# B&R Automation Studio project 8238 (part 32)

#### _getTourLoadingData.st
```iecst
ACTION _getTourLoadingData:

	prg	:= 0;
	cat := 0;
	cus := 0;
	dst := 0;
	sp1 := 0;
	sp2 := 0;
	sp3 := 0;
	index 	:= 0;
	tourID := 0;

	error := 0;
	found := 0;
	//Set common parameters of the function.
	getParameterName.searchString := requestData;
	getParameterName.searchOffset := 0;
	getParameterName.searchEndProperty := STRING_DOLLAR;

	//Find the index
	getParameterName.searchPropertyName := '"displayId":';
	getParameterName.searchEndProperty := ',';
	getParameterName();
	IF getParameterName.status = ERR_OK THEN
		index := DINT_TO_UDINT(atoi(ADR(getParameterName.outputValue)));
		getParameterName.searchOffset := getParameterName.nextPosition;
	ELSE
		error := 1;
	END_IF;

	//Find the category
	getParameterName.searchPropertyName := '"cat":';
	getParameterName.searchEndProperty := ',';
	getParameterName();
	IF getParameterName.status = ERR_OK THEN
		cat := DINT_TO_UDINT(atoi(ADR(getParameterName.outputValue)));
		getParameterName.searchOffset := getParameterName.nextPosition;
	ELSE
		error := 2;
	END_IF;

	//Find the customer
	getParameterName.searchPropertyName := '"cus":';
	getParameterName.searchEndProperty := ',';
	getParameterName();
	IF getParameterName.status = ERR_OK THEN
		cus := DINT_TO_UDINT(atoi(ADR(getParameterName.outputValue)));
		getParameterName.searchOffset := getParameterName.nextPosition;
	ELSE
		error := 3;
	END_IF;

	//Find the tour
	getParameterName.searchPropertyName := '"tourId":';
	getParameterName.searchEndProperty := ',';
	getParameterName();
	IF getParameterName.status = ERR_OK THEN
		tourID := DINT_TO_UDINT(atoi(ADR(getParameterName.outputValue)));
		getParameterName.searchOffset := getParameterName.nextPosition;
	ELSE
		error := 4;
	END_IF;

	//Find the Program
	getParameterName.searchPropertyName := '"prg":';
	getParameterName.searchEndProperty := ',';
	getParameterName();
	IF getParameterName.status = ERR_OK THEN
		prg := DINT_TO_USINT(atoi(ADR(getParameterName.outputValue)));
		getParameterName.searchOffset := getParameterName.nextPosition;
	ELSE
		error := 5;
	END_IF;

	//Find the sp1
	getParameterName.searchPropertyName := '"sp1":';
	getParameterName.searchEndProperty := ',';
	getParameterName();
	IF getParameterName.status = ERR_OK THEN
		sp1 := DINT_TO_UINT(atoi(ADR(getParameterName.outputValue)));
		getParameterName.searchOffset := getParameterName.nextPosition;
	ELSE
		error := 6;
	END_IF;

	//Find the sp2
	getParameterName.searchPropertyName := '"sp2":';
	getParameterName.searchEndProperty := ',';
	getParameterName();
	IF getParameterName.status = ERR_OK THEN
		sp2 := DINT_TO_UINT(atoi(ADR(getParameterName.outputValue)));
		getParameterName.searchOffset := getParameterName.nextPosition;
	ELSE
		error := 7;
	END_IF;
	//Find the sp3
	getParameterName.searchPropertyName := '"sp3":';
	getParameterName.searchEndProperty := ',';
	getParameterName();
	IF getParameterName.status = ERR_OK THEN
		sp3 := DINT_TO_UINT(atoi(ADR(getParameterName.outputValue)));
		getParameterName.searchOffset := 0;//getParameterName.nextPosition;
	ELSE
		error := 8;
	END_IF;

	//Find the program
	getParameterName.searchPropertyName := '"dst":';
	getParameterName.searchEndProperty := ',';
	getParameterName();
	IF getParameterName.status = ERR_OK THEN
		dst := DINT_TO_USINT(atoi(ADR(getParameterName.outputValue)));
		IF (index <= MAX_DISPLAYS) THEN
			found := found + 1;
			bag ACCESS ADR(LiveData_Recv[index].Bag);
			bag.Cat := cat;
			bag.Prg := prg;
			bag.Cus := cus;
			bag.Dst := dst;
			LiveData_Recv[index].Setpoints.SP1 := sp1 * 10;
			LiveData_Recv[index].Setpoints.SP2:= sp2 * 10;
			LiveData_Recv[index].Setpoints.SP3 := sp3 * 10;
			//bag.Tour := tourID;
		ELSE
			error := 99;
			overRideData.responseHeader.status := '404 Not Found';
			responseData := 'Unknown display';
			httpServer.responseDataLen := LEN(responseData);
		END_IF;
	ELSE
		error := 10;
	END_IF;

	sendResponse := (found > 0);
	errorResponse := (error > 0);

END_ACTION
```

#### _getTourLoadingSubmit.st
```iecst
ACTION _getTourLoadingSubmit:

	prg	:= 0;
	cat := 0;
	cus := 0;
	dst := 0;
	sp1 := 0;
	sp2 := 0;
	sp3 := 0;
	index 	:= 0;
	tourID := 0;

	error := 0;
	found := 0;
	//Set common parameters of the function.
	getParameterName.searchString := requestData;
	getParameterName.searchOffset := 0;
	getParameterName.searchEndProperty := STRING_DOLLAR;

	//Find the index
	getParameterName.searchPropertyName := '"displayId":';
	getParameterName.searchEndProperty := ',';
	getParameterName();
	IF getParameterName.status = ERR_OK THEN
		index := DINT_TO_UDINT(atoi(ADR(getParameterName.outputValue)));
		getParameterName.searchOffset := getParameterName.nextPosition;
	ELSE
		error := 1;
	END_IF;

	//Find the category
	getParameterName.searchPropertyName := '"cat":';
	getParameterName.searchEndProperty := ',';
	getParameterName();
	IF getParameterName.status = ERR_OK THEN
		cat := DINT_TO_UDINT(atoi(ADR(getParameterName.outputValue)));
		getParameterName.searchOffset := getParameterName.nextPosition;
	ELSE
		error := 2;
	END_IF;

	//Find the customer
	getParameterName.searchPropertyName := '"cus":';
	getParameterName.searchEndProperty := ',';
	getParameterName();
	IF getParameterName.status = ERR_OK THEN
		cus := DINT_TO_UDINT(atoi(ADR(getParameterName.outputValue)));
		getParameterName.searchOffset := getParameterName.nextPosition;
	ELSE
		error := 3;
	END_IF;

	//Find the tour
	getParameterName.searchPropertyName := '"tourId":';
	getParameterName.searchEndProperty := ',';
	getParameterName();
	IF getParameterName.status = ERR_OK THEN
		tourID := DINT_TO_UDINT(atoi(ADR(getParameterName.outputValue)));
		getParameterName.searchOffset := getParameterName.nextPosition;
	ELSE
		error := 4;
	END_IF;

	//Find the Program
	getParameterName.searchPropertyName := '"prg":';
	getParameterName.searchEndProperty := ',';
	getParameterName();
	IF getParameterName.status = ERR_OK THEN
		prg := DINT_TO_USINT(atoi(ADR(getParameterName.outputValue)));
		getParameterName.searchOffset := getParameterName.nextPosition;
	ELSE
		error := 5;
	END_IF;

	//Find the sp1
	getParameterName.searchPropertyName := '"sp1":';
	getParameterName.searchEndProperty := ',';
	getParameterName();
	IF getParameterName.status = ERR_OK THEN
		sp1 := DINT_TO_UINT(atoi(ADR(getParameterName.outputValue)));
		getParameterName.searchOffset := getParameterName.nextPosition;
	ELSE
		error := 6;
	END_IF;

	//Find the sp2
	getParameterName.searchPropertyName := '"sp2":';
	getParameterName.searchEndProperty := ',';
	getParameterName();
	IF getParameterName.status = ERR_OK THEN
		sp2 := DINT_TO_UINT(atoi(ADR(getParameterName.outputValue)));
		getParameterName.searchOffset := getParameterName.nextPosition;
	ELSE
		error := 7;
	END_IF;
	//Find the sp3
	getParameterName.searchPropertyName := '"sp3":';
	getParameterName.searchEndProperty := ',';
	getParameterName();
	IF getParameterName.status = ERR_OK THEN
		sp3 := DINT_TO_UINT(atoi(ADR(getParameterName.outputValue)));
		getParameterName.searchOffset := 0;//getParameterName.nextPosition;
	ELSE
		error := 8;
	END_IF;

	//Find the program
	getParameterName.searchPropertyName := '"dst":';
	getParameterName.searchEndProperty := ',';
	getParameterName();
	IF getParameterName.status = ERR_OK THEN
		dst := DINT_TO_USINT(atoi(ADR(getParameterName.outputValue)));
		IF (index <= MAX_DISPLAYS) THEN
			found := found + 1;
			bag ACCESS ADR(LiveData_Recv[index].Bag);
			bag.Cat := cat;
			bag.Prg := prg;
			bag.Cus := cus;
			bag.Dst := dst;
			LiveData_Recv[index].Setpoints.SP1 := sp1 * 10;
			LiveData_Recv[index].Setpoints.SP2:= sp2 * 10;
			LiveData_Recv[index].Setpoints.SP3 := sp3 * 10;
			LiveData_Recv[index].Submit_Loading := 1;

			//bag.Tour := tourID;
		ELSE
			error := 99;
			overRideData.responseHeader.status := '404 Not Found';
			responseData := 'Unknown display';
			httpServer.responseDataLen := LEN(responseData);
		END_IF;
	ELSE
		error := 10;
	END_IF;

	sendResponse := (found > 0);
	errorResponse := (error > 0);

END_ACTION
```

#### Types.typ - Local data types
```iecst
TYPE
	overRide_typ : 	STRUCT  (** OverRide Data to override default setting*)
		responseDataLen : UDINT;
		responseHeader : httpResponseHeader_t;
	END_STRUCT;
END_TYPE
```

#### LocalFunctions.fun
```iecst
FUNCTION_BLOCK httpGetParameter (*FUB to Get parameter values set in URI or BODY...*) (*$GROUP=User,$CAT=User,$GROUPICON=User.png,$CATICON=User.png*)
	VAR_INPUT
		searchPropertyName : STRING[50]; (*StringValue of propery or name to match*)
		searchEndProperty : STRING[50]; (*String Character or value to show end of property value -- DEFAULT & *)
		searchOffset : UINT; (*Offset can be set to skip searching begining of string if not required*)
		searchString : STRING[500];
	END_VAR
	VAR_OUTPUT
		outputValue : STRING[100]; (*String Value found*)
		status : UINT;
		nextPosition : UINT;
	END_VAR
	VAR
		matchString : STRING[50];
		inputData : ARRAY[0..499] OF USINT;
		endIndex : INT;
		startPosition : INT;
		n : INT;
		compare : DINT;
		length : UINT;
		startoffset : UINT;
		search : STRING[50];
	END_VAR
END_FUNCTION_BLOCK
```

#### httpGetParameter.st
```iecst
(* FUB to Get parameter values set in URI or BODY... *)
FUNCTION_BLOCK httpGetParameter
	status := ERR_FUB_BUSY;
// Get the function Name from the URI
//Use the string length of the service name	+
	memset(ADR(outputValue),0,SIZEOF(outputValue));
	matchString := searchPropertyName;
	strcpy(ADR(inputData[0]),ADR(searchString));
	startoffset := searchOffset;
	endIndex := LEN(searchString);
	startPosition := 16#FFF;
	IF endIndex > startoffset THEN
		FOR n := startoffset TO endIndex DO
			memcpy(ADR(search),ADR(inputData[n]),LEN(matchString));
			compare := 	strcmp(ADR(search),ADR(matchString));
			IF (compare = 0) THEN
				startPosition := n + LEN(matchString);
				EXIT;
			END_IF;
		END_FOR;
	ELSE
		status := 100;
	END_IF;

	IF (startPosition <> 16#FFF) THEN
		//Get the End Position
		matchString := searchEndProperty;
		memset(ADR(search),0,SIZEOF(search));
		startoffset := startPosition;
		IF endIndex >= startoffset THEN
			FOR n := startoffset TO endIndex DO
				memcpy(ADR(search),ADR(inputData[n]),LEN(matchString));
				compare := 	strcmp(ADR(search),ADR(matchString));
				length := n - startPosition;
				IF (compare = 0) THEN
					EXIT;
				END_IF;
			END_FOR;
			outputValue := MID(searchString,length,startPosition + 1);
			nextPosition := startPosition + length;
			status := ERR_OK;
		ELSE
			status := 102;
		END_IF;
	ELSE
		outputValue := '';
		nextPosition := 0;
		status := 101;
	END_IF;

END_FUNCTION_BLOCK
```

#### _updateVarByName.st
```iecst
//0, 15// Derived data types Data types declared with the construction TYPE...END_TYPE [1], [2]
//1:// BOOL 8-bit containing a boolean value FALSE=0 OR TRUE=1
//2:// SINT 8-bit signed integer
//3:// INT 16-bit signed integer
//4:// DINT 32-bit signed integer
//5:// USINT 8-bit unsigned integer
//6:// UINT 16-bit unsigned integer
//7:// UDINT 32-bit unsigned integer
//8:// REAL 32-bit floating point number
//9:// STRING Variable-length single-byte character string
//10:// ULINT 	64-bit unsigned integer
//11:// DATE_AND_TIME 32-bit date in seconds since 01/01/1970 00:00:00
//12:// TIME 32-bit time in ms
//13:// DATE 32-bit date (only)
//14:// LREAL 64-bit floating point number
//16:// TIME_OF_DAY 32-bit time OF day (only)
//17:// BYTE 	Bit string OF length 8
//18:// WORD Bit string OF length 16
//19:// DWORD Bit string OF length 32
//20:// LWORD Bit string OF length 64
//21:// WSTRING Variable-length double-byte character string
//23:// LINT 	64-bit signed integer

ACTION _updateVarByName:

//{"varName":"xxx","value":10}
//{"varName":"xxx","value":"stringValue"}
scanCount := 0;
WHILE (scanCount <= 19) AND NOT sendResponse AND NOT errorResponse DO
	scanCount := scanCount + 1; //Supercharge peformance by doing 20 scans per cycle

	CASE setValue OF

		0:// init search vars
			searchOffset := 0;
			//Create a FIFO to write our values into so we can commit them on success!!
			arrayEnd := FIND(requestData,'}]');// Be sure to check for end ] or we could get errors updating arrays.
			error := 0;
			setValue := 1;
			pos1 := 0;
			pos2 := 0;

		1:// create fifo to write data into.
			createFifo.enable := 1;
			createFifo.mode := fifoMODE_WRITE_UNTIL_FULL;
			createFifo.size := LEN(requestData);
			createFifo.pFifo := ADR('update-by-name-list');
			createFifo();
			IF (createFifo.status = ERR_OK) THEN
				setValue := 4;
			ELSIF (createFifo.status = fifoERR_FIFO_ALREADY_EXISTS) THEN
				setValue := 2;
			ELSIF (createFifo.status <> ERR_FUB_BUSY) THEN
				setValue := 100;
				status := 94;
			END_IF;

		2:// get ident if fifo already exists
			fi_status := fifoGetIdent(createFifo.pFifo,ADR(createFifo.ident));
			IF fi_status = ERR_OK THEN
				setValue := 3;
			ELSE
				setValue := 100;
				status := 94;
			END_IF;

		3:// Clear the FIFO if it already exists
			clearFifo.enable := 1;
			clearFifo.ident := createFifo.ident;
			clearFifo();
			IF clearFifo.status = ERR_OK THEN
				setValue := 4;
			ELSIF (clearFifo.status <> ERR_FUB_BUSY) THEN
				setValue := 100;
				status := 94;
			END_IF;

		4:// Validate the json, make sure if we have a [
			IF (arrayEnd > 0) THEN
				IF FIND(requestData,'[{') > 0 THEN
					setValue := 5; //Array start and end found
				ELSE
					setValue := 100;
					status := 95;
				END_IF;
			ELSE
				IF FIND(requestData,'[{') = 0 THEN
					setValue := 5; //Array start and end not found
				ELSE
					setValue := 100;
					status := 95;
				END_IF;
			END_IF;

		5://find the order of the parameters in the request sting.
			found 	:= 0;
			getParameterName.searchString := requestData;
			IF (pos1 = 0) THEN
				pos1 := FIND(requestData,SEARCH_STRING_VAR_NAME);
				pos2 := FIND(requestData,SEARCH_STRING_VAR_VALUE);
			END_IF;
			IF (pos1 = 0) OR (pos2 = 0) THEN
				setValue := 100;
				status := 93;
			ELSIF (pos1 > pos2) THEN
				setValue := 6;
			ELSE
				setValue := 8;
			END_IF;

		6:// find the value first
			value 	:= '';
			isString := 0;
			getParameterName.searchPropertyName := SEARCH_STRING_VAR_VALUE;
			getParameterName.searchEndProperty := ',';
			getParameterName.searchOffset := searchOffset;
			getParameterName();
			IF getParameterName.status = ERR_OK THEN
				searchOffset := getParameterName.nextPosition;
				//If we have been passed a string remove the ""
				IF LEFT(getParameterName.outputValue,1) = '"' THEN
					isString := 1;
					value := MID(getParameterName.outputValue,(LEN(getParameterName.outputValue) - 2),2);
				ELSE
					value := getParameterName.outputValue;
				END_IF;
				setValue := 7;
			ELSE
				setValue := 100;
				status := 2;
			END_IF;

		7:// find the name 2nd
			varName := '';
			found 	:= 0;
			//Set common parameters of the function.

			getParameterName.searchOffset := searchOffset;
			//Find the id
			getParameterName.searchPropertyName := SEARCH_STRING_VAR_NAME;
			getParameterName.searchEndProperty := '"';
			getParameterName();
			IF getParameterName.status = ERR_OK THEN
				varName := getParameterName.outputValue;
				searchOffset := getParameterName.nextPosition;
				setValue := 10;
			ELSE
				setValue := 100;
				status := 1;
			END_IF;

		8:// find the first param

			varName := '';
			getParameterName.searchOffset := searchOffset;
			//Find the id
			getParameterName.searchPropertyName := SEARCH_STRING_VAR_NAME;
			getParameterName.searchEndProperty := '"';
			getParameterName();
			IF getParameterName.status = ERR_OK THEN
				varName := getParameterName.outputValue;
				searchOffset := getParameterName.nextPosition;
				setValue := 9;
			ELSE
				setValue := 100;
				status := 1;
			END_IF;

		9:// find the 2nd param
			value 	:= '';
			isString := 0;
			getParameterName.searchPropertyName := SEARCH_STRING_VAR_VALUE;
			getParameterName.searchEndProperty := '}';
			getParameterName.searchOffset := searchOffset;
			getParameterName();
			IF getParameterName.status = ERR_OK THEN
				searchOffset := getParameterName.nextPosition;
				//If we have been passed a string remove the ""
				IF LEFT(getParameterName.outputValue,1) = '"' THEN
					isString := 1;
					value := MID(getParameterName.outputValue,(LEN(getParameterName.outputValue) - 2),2);
				ELSE
					value := getParameterName.outputValue;
				END_IF;
				setValue := 10;
			ELSE
				setValue := 100;
				status := 2;
			END_IF;

		10: //get the ident

			//status := PV_ident(ADR(varName),1,0,ADR(ident));
			status := PV_xgetadr(ADR(varName),ADR(pv_adr),ADR(pv_len));
			IF (status = ERR_OK) THEN
				setValue := 11;
			ELSIF (status <> ERR_FUB_BUSY) THEN
				IF (status = 14710) THEN
					overRideData.responseHeader.status := '404 Not Found';
					responseData := 'PV Not found';
					httpServer.responseDataLen := LEN(responseData);
				END_IF;
				setValue := 100;//
			END_IF;

		11: // Get the data type so we can scale correctly
			status := PV_ninfo(ADR(varName),ADR(pv_type),ADR(pv_length),ADR(pv_dimension));
			IF (status = ERR_OK) THEN
				setValue := 12;
			ELSIF (status <> ERR_FUB_BUSY) THEN
				setValue := 100;//
			END_IF;

		12: // Found update the value
			//Type 0 or 15 is part of a type not a var name.
			//We must also check the dimension is 1 or we are trying to update the root of an array.
			//TEMP INCASE OF MALFORM JSON
			//			IF (isString AND (pv_type <> 9)) THEN
			//				isString := 0;
			//			END_IF;

			stringCheck := (NOT isString AND (pv_type <> 9)) OR (isString AND (pv_type = 9)); // We have to modify this if we want to support strings other than STRING
			IF (pv_dimension = 1) AND stringCheck THEN
				num_Val := atoi(ADR(value));
				CASE pv_type OF
					0,15:// Derived data types Data types declared with the construction TYPE...END_TYPE [1], [2]
						status := 99;
						setValue := 100;
					1:// BOOL
						IF (num_Val >= 0) AND (num_Val <= 1) THEN
							pData := ADR(num_Val);
							//memcpy(pv_adr,ADR(num_Val),pv_length);
							found := 1;
						ELSE
							status := 96;
							setValue := 100;
						END_IF;
					2:// SINT
						IF (num_Val >= -128) AND (num_Val <= 16#7F) THEN
							pData := ADR(num_Val);
							//memcpy(pv_adr,ADR(num_Val),pv_length);
							found := 1;
						ELSE
							status := 96;
							setValue := 100;
						END_IF;
					3:// INT
						IF (num_Val >= -32768) AND (num_Val <= 16#7FFF) THEN
							pData := ADR(num_Val);
							//memcpy(pv_adr,ADR(num_Val),pv_length);
							found := 1;
						ELSE
							status := 96;
							setValue := 100;
						END_IF;
					4:// DINT
						IF (num_Val >= -2147483648) AND (num_Val <= 16#7FFFFFFF) THEN
							pData := ADR(num_Val);
							//memcpy(pv_adr,ADR(num_Val),pv_length);
							found := 1;
						ELSE
							status := 96;
							setValue := 100;
						END_IF;

					5: //USINT
						IF (num_Val >= 0) AND (num_Val <= 16#FF) THEN
							pData := ADR(num_Val);
							//memcpy(pv_adr,ADR(num_Val),pv_length);
							found := 1;
						ELSE
							status := 96;
							setValue := 100;
						END_IF;
					6:// UINT
						IF (num_Val >= 0) AND (num_Val <= 16#FFFF) THEN
							pData := ADR(num_Val);
							//memcpy(pv_adr,ADR(num_Val),pv_length);
							found := 1;
						ELSE
							status := 96;
							setValue := 100;
						END_IF;
					7: //UDINT
						IF (num_Val >= 0) AND (DINT_TO_UDINT(num_Val) <= 16#FFFF_FFFF) THEN  //
							pData := ADR(num_Val);
							//memcpy(pv_adr,ADR(num_Val),pv_length);
							found := 1;
						ELSE
							status := 96;
							setValue := 100;
						END_IF;

					8:// REAL 32-bit floating point number
						float_val := atof(ADR(value));
						IF (float_val >= -3.4E38) AND (float_val <= 3.4E38) THEN
							pData := ADR(float_val);
							//memcpy(pv_adr,ADR(float_val),pv_length);
							found := 1;
						ELSE
							status := 96;
							setValue := 100;
						END_IF;
						found := 1;

					9:// STRING Variable-length single-byte character string
						IF (LEN(value) <= pv_length) THEN
							memset(ADR(string_Val),0,pv_length);
							memcpy(ADR(string_Val),ADR(value),LEN(value));
							pData := ADR(string_Val);
							found := 1;
						ELSE
							status := 96;
							setValue := 100;
						END_IF;
					10..14,16..23:
						status := 98;
						setValue := 100;

				END_CASE;
			ELSIF NOT stringCheck THEN
				status := 97;
				setValue := 100;
			ELSE;
				status := 99;
				setValue := 100;
			END_IF;
			IF (found > 0) THEN
				setValue := 13;
			END_IF;

		13: // Add header data to the fifo
			data[0] := pv_adr;
			data[1] := pv_len;
			writeFifo.enable := 1;
			writeFifo.ident := createFifo.ident;
			writeFifo.pData := ADR(data[0]);
			writeFifo.size := 8;//
			writeFifo();
			IF (writeFifo.status = ERR_OK) THEN
				setValue := 14;
			ELSIF writeFifo.status <> ERR_FUB_BUSY THEN
				setValue := 100;
				status := 94;
			END_IF;

		14:// Add the actual data the fifo
			writeFifo.enable := 1;
			writeFifo.ident := createFifo.ident;
			writeFifo.pData := pData;
			writeFifo.size := pv_len;//
			writeFifo();
			IF (writeFifo.status = ERR_OK) THEN
				setValue := 20;
			ELSIF writeFifo.status <> ERR_FUB_BUSY THEN
				setValue := 100;
				status := 94;
			END_IF;

		20:// Check if we need to search again or complete the
			IF(arrayEnd <= 1) OR ((arrayEnd - searchOffset) < 5) THEN
				setValue := 30;
			ELSE //Search again
				setValue := 5;
			END_IF;

		30:// Process the results Read out the data header
			readFifo.enable := 1;
			readFifo.ident := createFifo.ident;
			readFifo.pData := ADR(data[0]);
			readFifo.size := 8;
			readFifo();
			IF (readFifo.status = ERR_OK) THEN
				pv_adr := data[0];
				pv_len := data[1];
				setValue := 31;
			ELSIF (readFifo.status = fifoERR_BUFFER_EMPTY) THEN
				setValue := 40;
			ELSIF readFifo.status <> ERR_FUB_BUSY THEN
				setValue := 100;
				status := 94;
			END_IF;

		31:// Process the results Read out the data
			readFifo.enable := 1;
			readFifo.ident := createFifo.ident;
			readFifo.pData := pv_adr;
			readFifo.size := pv_len;
			readFifo();
			IF (readFifo.status = ERR_OK) THEN
				setValue := 30; // Go back to iterate through the fifo
				//			ELSIF (readFifo.status = fifoERR_BUFFER_EMPTY) THEN
				//				setValue := 40;
			ELSIF readFifo.status <> ERR_FUB_BUSY THEN
				setValue := 100;
				status := 94;
			END_IF;

		40:// Delete the FIFO
			deleteFifo.enable := 1;
			deleteFifo.ident := createFifo.ident;
			deleteFifo();
			IF deleteFifo.status = ERR_OK THEN
				setValue := 90;
			ELSIF (deleteFifo.status <> ERR_FUB_BUSY) THEN
				setValue := 100;
				status := 94;
			END_IF;

		90:// Send the response

		100:// Error Step
			error := status;

			CASE status OF
				94:
					overRideData.responseHeader.status := '400 Bad Request';
					responseData := 'PLC FIFO Failure';
					httpServer.responseDataLen := LEN(responseData);

				95:
					overRideData.responseHeader.status := '400 Bad Request';
					responseData := 'Malformed JSON array';
					httpServer.responseDataLen := LEN(responseData);

				96:
					overRideData.responseHeader.status := '403 Forbidden';
					responseData := 'Value out of range';
					httpServer.responseDataLen := LEN(responseData);

				97:
					overRideData.responseHeader.status := '405 Method Not Allowed';
					responseData := 'You have sent a string to a numeric data type';
					httpServer.responseDataLen := LEN(responseData);

				98:
					overRideData.responseHeader.status := '405 Method Not Allowed';
					responseData := 'This data type is currently not supported';
					httpServer.responseDataLen := LEN(responseData);
				99:
					overRideData.responseHeader.status := '403 Forbidden';
					responseData := 'You have requested to update a structure part, or Array item without specifing the full path';
					httpServer.responseDataLen := LEN(responseData);
			END_CASE;

	END_CASE;

	sendResponse := (setValue = 90);
	errorResponse := (error > 0);
	//Configuration.Data.Belt[0].Alarm.General
	IF EDGEPOS(sendResponse) OR EDGEPOS(errorResponse) THEN
		setValue := 0;
	END_IF;
END_WHILE;

END_ACTION
```

#### _nedlinSetCustomer.st
```iecst
ACTION _nedlinSetCustomer:
	//{"stationId":1,"cus":25}
	IF (found = 0) AND (error = 0) THEN
		index := 0;
		cus := 0;

		error := 0;
		found := 0;
		//Set common parameters of the function.
		getParameterName.searchString := requestData;
		getParameterName.searchOffset := 0;
		getParameterName.searchEndProperty := STRING_DOLLAR;

		//Find the Index
		getParameterName.searchPropertyName := '"stationId":';
		getParameterName.searchEndProperty := ',';
		getParameterName();
		IF getParameterName.status = ERR_OK THEN
			index := DINT_TO_UDINT(atoi(ADR(getParameterName.outputValue)));
		ELSE
			error := 2;
		END_IF;

		//Find the customer
		getParameterName.searchPropertyName := '"cus":';
		getParameterName.searchEndProperty := ',';
		getParameterName();
		IF getParameterName.status = ERR_OK THEN
			cus := DINT_TO_USINT(atoi(ADR(getParameterName.outputValue)));
			IF (index >= 0) AND (index <= 1) THEN
				CSP[index].Customer := cus;
				found := found + 1;
			ELSE
				error := 99;
				overRideData.responseHeader.status := '404 Not Found';
				responseData := 'Index out of range';
				httpServer.responseDataLen := LEN(responseData);
			END_IF;
		ELSE
			error := 3;
		END_IF;
	END_IF;

	sendResponse := (found > 0);
	errorResponse := (error > 0);

END_ACTION
```

#### _resetCount.st
```iecst
ACTION _resetCount:
	//{"id":1}
	IF (found = 0) AND (error = 0) THEN
		index := 0;
		cus := 0;

		error := 0;
		found := 0;
		//Set common parameters of the function.
		getParameterName.searchString := requestData;
		getParameterName.searchOffset := 0;
		getParameterName.searchEndProperty := STRING_DOLLAR;

		//Find the Index
		getParameterName.searchPropertyName := '"id":';
		getParameterName.searchEndProperty := '}';
		getParameterName();
		IF getParameterName.status = ERR_OK THEN
			index := DINT_TO_UDINT(atoi(ADR(getParameterName.outputValue)));
			IF (index >= 0) AND (index <= MAX_STATIONS) THEN
				SortingBins.counting_frames[index].count := 0;
				found := found + 1;
			ELSE
				error := 99;
				overRideData.responseHeader.status := '404 Not Found';
				responseData := 'Index out of range';
				httpServer.responseDataLen := LEN(responseData);
			END_IF;

		ELSE
			error := 2;
		END_IF;
	END_IF;

	sendResponse := (found > 0);
	errorResponse := (error > 0);

END_ACTION
```

### HttpInstances.txt
```
List Of HTTP_Comm indexes

01: zzReportsHttp
02: SLX_Inteface
03: Configuration
04: OPCuA_Connect
05: Bag Maintenance
06:
07:
08:
09:
10:
11:
12:
13:
14:
15:
16:
17:
18:
19:
20:
```

### Program Logical/http_Lib/zzHttpDriver (IEC, version 3.00.8)

#### Types.typ - Local data types
```iecst
TYPE
	httpState_enum :
		(
		HTTP_CLIENT_WAIT_FOR_COMMAND := 0,
		HTTP_CLIENT_PROCESS_REQUEST := 1,
		HTTP_CLIENT_PROCESS_ENABLE := 2,
		HTTP_CLIENT_PROCESS_SEND := 3,
		HTTP_CLIENT_PROCESS_WAIT_RESP := 4,
		HTTP_CLIENT_PROCESS_RESPONSE := 5,
		HTTP_CLIENT_COMPLETE := 6,
		HTTP_CLIENT_ABORT := 99
		);
END_TYPE
```

#### Variables.var - Local variables
```iecst
VAR
	n : UINT;
	r : UINT;
	httpComm : REFERENCE TO http_comm_typ;
	ringBuffer : ARRAY[0..HTTP_MAX_COMM] OF UINT;
	sizeRingArray : UDINT;
	sizeRingData : UDINT;
	moveSize : UDINT;
	pUrl : UDINT;
	URL : STRING[500];
	pHost : UDINT;
	pResponseHeader : UDINT;
	pTempMem : UDINT;
	sizeTempMem : UDINT;
	pStatistics : UDINT;
	responseHeader : httpResponseHeader_t;
	http_Client : httpClient;
	Statistics : {REDUND_UNREPLICABLE} httpStatistics_t;
	emptyResponseHeader : httpResponseHeader_t;
	DebugErrCount : UDINT;
	pRequestHeader : UDINT;
	requestHeader : httpRequestHeader_t;
	remainingStringLen : DINT;
END_VAR
VAR CONSTANT
	BLANK_CHARACTER : STRING[80] := '';
END_VAR
VAR
	httpState : httpState_enum;
	retryCount : USINT;
	status : HTTP_Status_enum;
	lastError : STRING[60];
	replyCode : UINT;
	count : UDINT;
	testEnable : BOOL;
	testAbort : BOOL;
END_VAR
```

#### Main.st - Init, cyclic, exit code
```iecst
//V2.00.1- First Release of Version Control - Remove all unused code- Removed temp memory for recieve data as this helps when we get a "Invalid Character error"
//V2.00.2 -- ADD: New error handling if we do not recieve data when expected.
//V2.00.3 -- ADD: Add http reply code to the http data type so we don;t have to decode the string in the user tasks
//V3.00.1 -- CHANGE: TR 23/08/2019 - Convert the driver to a state machine
//V3.00.2 -- FIX: When writing to reports the status is being set as disabled causing repeated writes -- Comment out in HTTP_CLIENT_PROCESS_REQUEST and it works.. It makes no sense!!
//V3.00.3 -- FIX: Found solution to 3.02. The original state was being set to DISABLE so the proces step was exiting incorrectly.
//V3.00.4 -- FIX: Issue with certain errors getting stuck on the abort step.
//V3.00.5 -- FIX: 35560 error non more idents availble!!
//V3.00.6 -- FIX: URL Wasn;t not being cleared correctly
//V3.00.7 -- FIX: TCP ERROR could lock up the driver.
//V3.00.8 -- FIX: The way we were passing the http port mean that it was always being set to 0 reegardless of the default setting, when not using overwrite
PROGRAM _INIT
	//Use Static code now but change to config file later..
	HTTP_Config.Host := '10.8.4.220';
	HTTP_Config.Port := 0;
	httpComm ACCESS ADR(HTTP_Comm[0]);

	pUrl 							:= ADR(URL);
	pRequestHeader 					:= ADR(requestHeader);
	pResponseHeader 				:= ADR(responseHeader);
	pStatistics 					:= ADR(Statistics);
	pHost 							:= ADR(requestHeader.host);

	http_Client.pUri 				:= pUrl;
	http_Client.option 				:= httpOPTION_HTTP_11;
	http_Client.pHost 				:= pHost;
	http_Client.pRequestHeader 		:= pRequestHeader;
	http_Client.pResponseHeader 	:= pResponseHeader;
	http_Client.pStatistics 		:= pStatistics;

	//Configure RequestHeader
	requestHeader.protocol := DEFAULT_REQUEST_HEADER.protocol; //'HTTP/1.1';
	requestHeader.contentType := DEFAULT_REQUEST_HEADER.contentType;//'text/plain';
	requestHeader.connection := DEFAULT_REQUEST_HEADER.connection;//'close';
	requestHeader.keepAlive := DEFAULT_REQUEST_HEADER.keepAlive;//'max=100,timeout=5';

	sizeTempMem := 500000; //Allocate 500k of free memory
	TMP_alloc(sizeTempMem,ADR(pTempMem));

	ringBuffer[0] := 0;
	//Check for any requests that were being processed on shut down..
	FOR n := 1 TO HTTP_MAX_COMM DO
		IF HTTP_Comm[n].Status = HTTP_COMM_STATUS_IN_PROCESS THEN
			ringBuffer[0] := n;
		ELSIF HTTP_Comm[n].Status = HTTP_COMM_STATUS_IN_BUFFER THEN
			ringBuffer[n] := n;
		END_IF;
	END_FOR;
	_orderRing;
END_PROGRAM

PROGRAM _CYCLIC

	//Listen to requests and add to ring buffer.
	_ringBuffer;
	http_Client.send	:= EDGEPOS(httpState = HTTP_CLIENT_PROCESS_SEND );
	http_Client.abort	:= EDGEPOS(httpState = HTTP_CLIENT_ABORT);

	CASE httpState OF

		HTTP_CLIENT_WAIT_FOR_COMMAND: // Order the ring buffer and wait for a new command to be processed.
			http_Client.enable := 0;
			retryCount := 0;
			httpComm ACCESS ADR(HTTP_Comm[0]);
			//Wait for next command from ring buffer
			IF(ringBuffer[0] = 0) AND (ringBuffer[1] > 0) THEN
				ringBuffer[0] := ringBuffer[1];
				httpComm ACCESS ADR(HTTP_Comm[ringBuffer[0]]);
				httpComm.Status := HTTP_COMM_STATUS_IN_PROCESS;
				ringBuffer[1] := 0;
			ELSIF (ringBuffer[0] > 0) THEN
				httpState := HTTP_CLIENT_PROCESS_REQUEST;
			END_IF;

		HTTP_CLIENT_PROCESS_REQUEST:
			http_Client.enable := 0;

			replyCode := 0;
			status := HTTP_COMM_STATUS_IN_PROCESS;
			lastError := '';

			httpComm ACCESS ADR(HTTP_Comm[ringBuffer[0]]);

			//brsmemcpy(ADR(URL),ADR(BLANK_CHARACTER),SIZEOF(URL));
			brsmemset(ADR(URL),0,SIZEOF(URL));
			//URL := '';
			brsmemcpy(ADR(URL),httpComm.Command.Cmd_URL.Adr,httpComm.Command.Cmd_URL.Size);
			responseHeader := emptyResponseHeader;

			//Check for any overwrite of the host or header
			IF httpComm.Overwrite.RequestHeader THEN
				requestHeader.protocol 		:= httpComm.Overwrite.RequestHeader_Data.protocol;
				requestHeader.contentType 	:= httpComm.Overwrite.RequestHeader_Data.contentType;
				requestHeader.connection 	:= httpComm.Overwrite.RequestHeader_Data.connection;
				requestHeader.keepAlive 	:= httpComm.Overwrite.RequestHeader_Data.keepAlive;
			ELSE
				requestHeader.protocol 		:= DEFAULT_REQUEST_HEADER.protocol; //'HTTP/1.1';
				requestHeader.contentType 	:= DEFAULT_REQUEST_HEADER.contentType;//'text/plain';
				requestHeader.connection 	:= DEFAULT_REQUEST_HEADER.connection;//'close';
				requestHeader.keepAlive 	:= DEFAULT_REQUEST_HEADER.keepAlive;//'max=100,timeout=5';
			END_IF;
			IF httpComm.Overwrite.Host THEN
				requestHeader.host 		:= httpComm.Overwrite.Host_Config.Host;
				http_Client.hostPort  	:= httpComm.Overwrite.Host_Config.Port;
			ELSE
				requestHeader.host 		:= HTTP_Config.Host;
				http_Client.hostPort 	:= HTTP_Config.Port;
			END_IF;

			requestHeader.contentLength 	:= httpComm.Command.Body_Data.Size;
			http_Client.method 				:= httpComm.Command.Method;
			http_Client.pRequestData 		:= httpComm.Command.Body_Data.Adr;
			http_Client.requestDataLen 		:= httpComm.Command.Body_Data.Size;

			IF (httpComm.Command.ResponseData.Adr > 0) AND (httpComm.Command.ResponseData.Size > 0) THEN
				http_Client.pResponseData 	:= httpComm.Command.ResponseData.Adr;
				http_Client.responseDataSize := httpComm.Command.ResponseData.Size;
			ELSE
				http_Client.pResponseData := pTempMem;
				http_Client.responseDataSize := sizeTempMem;
			END_IF;
			IF (http_Client.status = ERR_FUB_ENABLE_FALSE) AND (http_Client.phase = httpPHASE_NOT_CONNECTED) THEN
				httpState := HTTP_CLIENT_PROCESS_ENABLE;
			END_IF;

		HTTP_CLIENT_PROCESS_ENABLE:
			http_Client.enable := 1;
			IF (http_Client.status = ERR_OK) THEN
				CASE http_Client.phase OF
					httpPHASE_NOT_CONNECTED,httpPHASE_WAITING:
						httpState := HTTP_CLIENT_PROCESS_SEND;

					httpPHASE_SENDING,httpPHASE_RECEIVING:
						httpState := HTTP_CLIENT_PROCESS_WAIT_RESP;

					httpPHASE_RECEIVED:
						httpState := HTTP_CLIENT_PROCESS_SEND; // Received is the left over from the last successful send.
				END_CASE;
			END_IF;

		HTTP_CLIENT_PROCESS_SEND:
			http_Client.enable := 1;
			IF (http_Client.phase = httpPHASE_SENDING) THEN
				httpState := HTTP_CLIENT_PROCESS_WAIT_RESP;
			ELSIF (http_Client.status <> ERR_OK) AND (http_Client.status <> ERR_FUB_BUSY) THEN
				httpState := HTTP_CLIENT_ABORT;
			ELSIF (http_Client.phase = httpPHASE_RECEIVED) AND (http_Client.httpStatus > 0) THEN
				httpState := HTTP_CLIENT_PROCESS_RESPONSE;
			END_IF;

		HTTP_CLIENT_PROCESS_WAIT_RESP:
			http_Client.enable := 1;
			IF (http_Client.phase = httpPHASE_RECEIVED) THEN
				httpState := HTTP_CLIENT_PROCESS_RESPONSE;
			ELSIF (http_Client.status <> ERR_OK) AND (http_Client.status <> ERR_FUB_BUSY) THEN
				httpState := HTTP_CLIENT_ABORT;
			END_IF;

		HTTP_CLIENT_PROCESS_RESPONSE:
			http_Client.enable := 1;
			IF (http_Client.status = ERR_OK) THEN
				replyCode := http_Client.httpStatus;
				CASE http_Client.httpStatus OF
					200..207:
						IF (responseHeader.contentLength > 0) THEN
							IF (responseHeader.contentLength <= httpComm.Command.ResponseData.Size) THEN
								status := HTTP_COMM_STATUS_COMPLETE;
							ELSE
								status := HTTP_COMM_STATUS_ERROR;
								lastError := 'Response data area to small';
							END_IF;
						ELSIF ((httpComm.Command.Method = httpMETHOD_POST) OR (httpComm.Command.Method = httpMETHOD_PUT)) THEN
							status := HTTP_COMM_STATUS_COMPLETE;
						END_IF;
					300..307:
						//Implementation not done
						status := HTTP_COMM_STATUS_ERROR;
						lastError := responseHeader.status;
					400..426: //Errors
						status := HTTP_COMM_STATUS_ERROR;
						lastError := responseHeader.status;
					500..510://Server Errors
						status	:= HTTP_COMM_STATUS_ERROR;
						lastError 	:= responseHeader.status;
					ELSE
						httpState 	:= HTTP_CLIENT_ABORT;
				END_CASE;
			ELSIF (http_Client.status = httpERR_BUFFER_SIZE) THEN	// Response buffer is too small -- Abort and try again with temp memory area

			ELSIF (http_Client.status <> ERR_FUB_BUSY) THEN	//http client failure.
				itoa(http_Client.status,ADR(lastError));
				httpState := HTTP_CLIENT_ABORT;
			END_IF;

			IF (status <> HTTP_COMM_STATUS_IN_PROCESS) THEN
				httpState := HTTP_CLIENT_COMPLETE;
			END_IF;

		HTTP_CLIENT_COMPLETE:
			count := count + 1;
			http_Client.enable := 0;
			httpComm.Status := status;
			httpComm.LastError := lastError;
			httpComm.ReplyCode := replyCode;
			ringBuffer[0] := 0;
			httpState := HTTP_CLIENT_WAIT_FOR_COMMAND;

		HTTP_CLIENT_ABORT:
			http_Client.enable := 1;

			IF ((http_Client.status = ERR_OK) AND NOT http_Client.abort) THEN
				IF (http_Client.phase = httpPHASE_WAITING) OR (http_Client.phase = httpPHASE_NOT_CONNECTED)  THEN
					IF (retryCount > 0) THEN
						httpState := HTTP_CLIENT_COMPLETE;
						status := HTTP_COMM_STATUS_ERROR;
					ELSE
						retryCount := 1;
						httpState := HTTP_CLIENT_PROCESS_REQUEST;
					END_IF;
				ELSIF (http_Client.phase = httpPHASE_RECEIVED) THEN //???
					IF (retryCount > 0) THEN
						httpState := HTTP_CLIENT_COMPLETE;
						status := HTTP_COMM_STATUS_ERROR;
					ELSE
						retryCount := 1;
						httpState := HTTP_CLIENT_PROCESS_REQUEST;
					END_IF;
				END_IF;
			END_IF;
	END_CASE;

	http_Client();

END_PROGRAM
PROGRAM _EXIT
	WHILE (http_Client.status <> ERR_OK) DO
		http_Client.enable := 1;
		http_Client.abort := 1;
		http_Client();
	END_WHILE;

END_PROGRAM
```

#### _ringBuffer.st
```iecst
ACTION _ringBuffer:

	//Listen to new comm events..
	FOR n := 0 TO HTTP_MAX_COMM DO
		//httpComm ACCESS ADR(HTTP_Comm[n]);
		//There is an active comm that is not in the buffer...
		IF (HTTP_Comm[n].Status = HTTP_COMM_STATUS_ACTIVE_WAIT_BUF) THEN
			_addToRing;	//Add to the next avaible space in the ring buffer.
		END_IF;
	END_FOR;

	//Update the ring to ensure we clear any comms that are in error or complete.
	//If a comm is in error, it should be upto the requesting task to clear the error and retry to comm..
	_orderRing;

END_ACTION
```

#### _addToRing.st
```iecst
ACTION _addToRing:
	FOR r := 1 TO HTTP_MAX_COMM DO
		IF (ringBuffer[r] = 0) THEN
			ringBuffer[r] := n;
			HTTP_Comm[n].Status := HTTP_COMM_STATUS_IN_BUFFER;
			EXIT;
		END_IF;
	END_FOR;
END_ACTION
```

#### _orderRing.st
```iecst
ACTION _orderRing:
	//Only loop from position 1 as 0 will be active..
	FOR n := 1 TO HTTP_MAX_COMM DO
		r := ringBuffer[n];
		//If the comm is in not in the queue, or in process then remove it from the queue.
		IF (HTTP_Comm[r].Status <> HTTP_COMM_STATUS_IN_BUFFER)  THEN
			ringBuffer[n] := 0;
		END_IF;
	END_FOR;
	//Shuffle List
	FOR n:= 1 TO (HTTP_MAX_COMM - 1)DO
		IF ringBuffer[n] = 0 THEN
			sizeRingArray := SIZEOF(ringBuffer);
			sizeRingData := SIZEOF(ringBuffer[0]);
			moveSize := (sizeRingArray - ((n+1)*sizeRingData));
			memcpy(ADR(ringBuffer[n]),ADR(ringBuffer[n + 1]),moveSize);
			ringBuffer[HTTP_MAX_COMM] := 0;
		END_IF;
	END_FOR
END_ACTION
```

### Program Logical/LOADCELLS (IEC, version 1.00.1) - LOADCELLS

#### LOADCELLS.st
```iecst
(********************************************************************
 * Program: LOADCELLS
 * File: LOADCELLS.st
 ********************************************************************)
PROGRAM _CYCLIC
(********************************************************************
* ALL SERVOS WITHIN A GROUP MUST HAVE ASCENDING RAIL ID'S
 ********************************************************************)
//	weight1 := DINT_TO_UINT(ABS(WeightRaw[1301].Wgt_Channel_1)/100);
//	weight2 := DINT_TO_UINT(ABS(WeightRaw[1302].Wgt_Channel_1)/100);
//	weight3 := DINT_TO_UINT(ABS(WeightRaw[1303].Wgt_Channel_1)/100);
//	weight4 := DINT_TO_UINT(ABS(WeightRaw[1304].Wgt_Channel_1)/100);
//	weight5 := DINT_TO_UINT(ABS(WeightRaw[1305].Wgt_Channel_1)/100);
//	weight6 := DINT_TO_UINT(ABS(WeightRaw[1306].Wgt_Channel_1)/100);
//	weight7 := DINT_TO_UINT(ABS(WeightRaw[1307].Wgt_Channel_1)/100);
//	weight8 := DINT_TO_UINT(ABS(WeightRaw[1308].Wgt_Channel_1)/100);
//	weight9 := DINT_TO_UINT(ABS(WeightRaw[1309].Wgt_Channel_1)/100);
//	weight10 := DINT_TO_UINT(ABS(WeightRaw[1310].Wgt_Channel_1)/100);
//	weight11 := DINT_TO_UINT(ABS(WeightRaw[1311].Wgt_Channel_1)/100);
//	weight12 := DINT_TO_UINT(ABS(WeightRaw[1312].Wgt_Channel_1)/100);
//	weight13 := DINT_TO_UINT(ABS(WeightRaw[1313].Wgt_Channel_1)/100);
//	weight14 := DINT_TO_UINT(ABS(WeightRaw[1314].Wgt_Channel_1)/100);
//	weight15 := DINT_TO_UINT(ABS(WeightRaw[1315].Wgt_Channel_1)/100);
//	weight16 := DINT_TO_UINT(ABS(WeightRaw[1316].Wgt_Channel_1)/100);
//	weight17 := DINT_TO_UINT(ABS(WeightRaw[1317].Wgt_Channel_1)/100);
//	weight18 := DINT_TO_UINT(ABS(WeightRaw[1318].Wgt_Channel_1)/100);
//	weight19 := DINT_TO_UINT(ABS(WeightRaw[1319].Wgt_Channel_1)/100);
//	weight20 := DINT_TO_UINT(ABS(WeightRaw[1320].Wgt_Channel_1)/100);
//	weight21 := DINT_TO_UINT(ABS(WeightRaw[1321].Wgt_Channel_1)/100);
//	weight22 := DINT_TO_UINT(ABS(WeightRaw[1322].Wgt_Channel_1)/100);
//	weight23 := DINT_TO_UINT(ABS(WeightRaw[1323].Wgt_Channel_1)/100);
//	weight24 := DINT_TO_UINT(ABS(WeightRaw[1324].Wgt_Channel_1)/100);
//	weight25 := DINT_TO_UINT(ABS(WeightRaw[1325].Wgt_Channel_1)/100);
//	weight26 := DINT_TO_UINT(ABS(WeightRaw[1302].Wgt_Channel_1)/100);
//	weight27 := DINT_TO_UINT(ABS(WeightRaw[1327].Wgt_Channel_1)/100);
//	weight28 := DINT_TO_UINT(ABS(WeightRaw[1304].Wgt_Channel_1)/100);
//	weight29 := DINT_TO_UINT(ABS(WeightRaw[1329].Wgt_Channel_1)/100);
//	weight30 := DINT_TO_UINT(ABS(WeightRaw[1306].Wgt_Channel_1)/100);
//	weight31 := DINT_TO_UINT(ABS(WeightRaw[1331].Wgt_Channel_1)/100);
//	weight32 := DINT_TO_UINT(ABS(WeightRaw[1308].Wgt_Channel_1)/100);
//	weight33 := DINT_TO_UINT(ABS(WeightRaw[1333].Wgt_Channel_1)/100);
//	weight34 := DINT_TO_UINT(ABS(WeightRaw[1310].Wgt_Channel_1)/100);
//	weight35 := DINT_TO_UINT(ABS(WeightRaw[1335].Wgt_Channel_1)/100);
//	weight36 := DINT_TO_UINT(ABS(WeightRaw[1312].Wgt_Channel_1)/100);
//	weight37 := DINT_TO_UINT(ABS(WeightRaw[1337].Wgt_Channel_1)/100);
//	weight38 := DINT_TO_UINT(ABS(WeightRaw[1314].Wgt_Channel_1)/100);
//	weight39 := DINT_TO_UINT(ABS(WeightRaw[1339].Wgt_Channel_1)/100);
//	weight40 := DINT_TO_UINT(ABS(WeightRaw[1316].Wgt_Channel_1)/100);
//	weight41 := DINT_TO_UINT(ABS(WeightRaw[1341].Wgt_Channel_1)/100);
//	weight42 := DINT_TO_UINT(ABS(WeightRaw[1318].Wgt_Channel_1)/100);
//	weight43 := DINT_TO_UINT(ABS(WeightRaw[1343].Wgt_Channel_1)/100);
//	weight44 := DINT_TO_UINT(ABS(WeightRaw[1320].Wgt_Channel_1)/100);
//	weight45 := DINT_TO_UINT(ABS(WeightRaw[1345].Wgt_Channel_1)/100);
//	weight46 := DINT_TO_UINT(ABS(WeightRaw[1322].Wgt_Channel_1)/100);
//	weight47 := DINT_TO_UINT(ABS(WeightRaw[1347].Wgt_Channel_1)/100);
//	weight48 := DINT_TO_UINT(ABS(WeightRaw[1324].Wgt_Channel_1)/100);
//	weight49 := DINT_TO_UINT(ABS(WeightRaw[1349].Wgt_Channel_1)/100);
//	weight50 := DINT_TO_UINT(ABS(WeightRaw[1349].Wgt_Channel_1)/100);
//	weight51 := DINT_TO_UINT(ABS(WeightRaw[1349].Wgt_Channel_1)/100);
//	weight52 := DINT_TO_UINT(ABS(WeightRaw[1352].Wgt_Channel_1)/100);
//	weight53 := DINT_TO_UINT(ABS(WeightRaw[1352].Wgt_Channel_1)/100);
//	weight54 := DINT_TO_UINT(ABS(WeightRaw[1352].Wgt_Channel_1)/100);
//	weight55 := DINT_TO_UINT(ABS(WeightRaw[1355].Wgt_Channel_1)/100);
//	weight56 := DINT_TO_UINT(ABS(WeightRaw[1355].Wgt_Channel_1)/100);
//	weight57 := DINT_TO_UINT(ABS(WeightRaw[1355].Wgt_Channel_1)/100);
//	weight58 := DINT_TO_UINT(ABS(WeightRaw[1358].Wgt_Channel_1)/100);
//	weight59 := DINT_TO_UINT(ABS(WeightRaw[1358].Wgt_Channel_1)/100);
//	weight60 := DINT_TO_UINT(ABS(WeightRaw[1368].Wgt_Channel_1)/100);
//	weight61 := DINT_TO_UINT(ABS(WeightRaw[1361].Wgt_Channel_1)/100);
//	weight62 := DINT_TO_UINT(ABS(WeightRaw[1361].Wgt_Channel_1)/100);
//	weight63 := DINT_TO_UINT(ABS(WeightRaw[1361].Wgt_Channel_1)/100);
//	weight64 := DINT_TO_UINT(ABS(WeightRaw[1364].Wgt_Channel_1)/100);
//	weight65 := DINT_TO_UINT(ABS(WeightRaw[1364].Wgt_Channel_1)/100);
//	weight66 := DINT_TO_UINT(ABS(WeightRaw[1364].Wgt_Channel_1)/100);
//	weight67 := DINT_TO_UINT(ABS(WeightRaw[1367].Wgt_Channel_1)/100);
//	weight68 := DINT_TO_UINT(ABS(WeightRaw[1367].Wgt_Channel_1)/100);
//	weight69 := DINT_TO_UINT(ABS(WeightRaw[1367].Wgt_Channel_1)/100);
//	weight70 := DINT_TO_UINT(ABS(WeightRaw[1370].Wgt_Channel_1)/100);
//	weight71 := DINT_TO_UINT(ABS(WeightRaw[1370].Wgt_Channel_1)/100);
//	weight72 := DINT_TO_UINT(ABS(WeightRaw[1370].Wgt_Channel_1)/100);
//	weight73 := DINT_TO_UINT(ABS(WeightRaw[1373].Wgt_Channel_1)/100);
//	weight74 := DINT_TO_UINT(ABS(WeightRaw[1373].Wgt_Channel_1)/100);
//	weight75 := DINT_TO_UINT(ABS(WeightRaw[1373].Wgt_Channel_1)/100);
//	weight76 := DINT_TO_UINT(ABS(WeightRaw[1376].Wgt_Channel_1)/100);
//	weight77 := DINT_TO_UINT(ABS(WeightRaw[1376].Wgt_Channel_1)/100);
//	weight78 := DINT_TO_UINT(ABS(WeightRaw[1376].Wgt_Channel_1)/100);
//	weight79 := DINT_TO_UINT(ABS(WeightRaw[1379].Wgt_Channel_1)/100);
//	weight80 := DINT_TO_UINT(ABS(WeightRaw[1379].Wgt_Channel_1)/100);
//	weight81 := DINT_TO_UINT(ABS(WeightRaw[1379].Wgt_Channel_1)/100);
//	weight82 := DINT_TO_UINT(ABS(WeightRaw[1382].Wgt_Channel_1)/100);
//	weight83 := DINT_TO_UINT(ABS(WeightRaw[1382].Wgt_Channel_1)/100);
//	weight84 := DINT_TO_UINT(ABS(WeightRaw[1382].Wgt_Channel_1)/100);
//	weight85 := DINT_TO_UINT(ABS(WeightRaw[1385].Wgt_Channel_1)/100);
//	weight86 := DINT_TO_UINT(ABS(WeightRaw[1385].Wgt_Channel_1)/100);
//	weight87 := DINT_TO_UINT(ABS(WeightRaw[1385].Wgt_Channel_1)/100);
//	weight88 := DINT_TO_UINT(ABS(WeightRaw[1388].Wgt_Channel_1)/100);
//	weight89 := DINT_TO_UINT(ABS(WeightRaw[1388].Wgt_Channel_1)/100);
//	weight90 := DINT_TO_UINT(ABS(WeightRaw[1388].Wgt_Channel_1)/100);
//	weight91 := DINT_TO_UINT(ABS(WeightRaw[1391].Wgt_Channel_1)/100);
//	weight92 := DINT_TO_UINT(ABS(WeightRaw[1391].Wgt_Channel_1)/100);
//	weight93 := DINT_TO_UINT(ABS(WeightRaw[1391].Wgt_Channel_1)/100);
//	weight94 := DINT_TO_UINT(ABS(WeightRaw[1394].Wgt_Channel_1)/100);
//	weight95 := DINT_TO_UINT(ABS(WeightRaw[1394].Wgt_Channel_1)/100);
//	weight96 := DINT_TO_UINT(ABS(WeightRaw[1394].Wgt_Channel_1)/100);
//	weight97 := DINT_TO_UINT(ABS(WeightRaw[1397].Wgt_Channel_1)/100);
//	weight98 := DINT_TO_UINT(ABS(WeightRaw[1397].Wgt_Channel_1)/100);
//	weight99 := DINT_TO_UINT(ABS(WeightRaw[1397].Wgt_Channel_1)/100);
//	weight100 := DINT_TO_UINT(ABS(WeightRaw[1600].Wgt_Channel_1)/100);
//	weight101 := DINT_TO_UINT(ABS(WeightRaw[1600].Wgt_Channel_1)/100);
//	weight102 := DINT_TO_UINT(ABS(WeightRaw[1600].Wgt_Channel_1)/100);
//	weight103 := DINT_TO_UINT(ABS(WeightRaw[1603].Wgt_Channel_1)/100);
//	weight104 := DINT_TO_UINT(ABS(WeightRaw[1603].Wgt_Channel_1)/100);
//	weight105 := DINT_TO_UINT(ABS(WeightRaw[1603].Wgt_Channel_1)/100);
//	weight106 := DINT_TO_UINT(ABS(WeightRaw[1606].Wgt_Channel_1)/100);
//	weight107 := DINT_TO_UINT(ABS(WeightRaw[1606].Wgt_Channel_1)/100);
//	weight108 := DINT_TO_UINT(ABS(WeightRaw[1606].Wgt_Channel_1)/100);
//	weight109 := DINT_TO_UINT(ABS(WeightRaw[1609].Wgt_Channel_1)/100);
//	weight110 := DINT_TO_UINT(ABS(WeightRaw[1609].Wgt_Channel_1)/100);
//	weight111 := DINT_TO_UINT(ABS(WeightRaw[1609].Wgt_Channel_1)/100);
//	weight112 := DINT_TO_UINT(ABS(WeightRaw[1612].Wgt_Channel_1)/100);
//	weight113 := DINT_TO_UINT(ABS(WeightRaw[1612].Wgt_Channel_1)/100);
//	weight114 := DINT_TO_UINT(ABS(WeightRaw[1612].Wgt_Channel_1)/100);
//	weight115 := DINT_TO_UINT(ABS(WeightRaw[1615].Wgt_Channel_1)/100);
//	weight116 := DINT_TO_UINT(ABS(WeightRaw[1615].Wgt_Channel_1)/100);
//	weight117 := DINT_TO_UINT(ABS(WeightRaw[1615].Wgt_Channel_1)/100);
//	weight118 := DINT_TO_UINT(ABS(WeightRaw[1618].Wgt_Channel_1)/100);
//	weight119 := DINT_TO_UINT(ABS(WeightRaw[1618].Wgt_Channel_1)/100);
//	weight120 := DINT_TO_UINT(ABS(WeightRaw[1618].Wgt_Channel_1)/100);
END_PROGRAM
```

#### Variables.var - not listed in the package file held
```iecst
VAR
	i : INT;
	testweight : UINT;
END_VAR
```

#### Main.st - not listed in the package file held
```iecst
(********************************************************************
 * Program: loadcells
 * File: loadcells.st
 ********************************************************************)
PROGRAM _INIT
//  FOR i := 1 TO 49 DO
//    loadcell_array[i].udp_data := ADR(loadcell_udp_array[i]);
//  END_FOR;

END_PROGRAM

PROGRAM _CYCLIC

	//==============================
	//	//Weights
	//==============================

	//Sorting
	IF NOT Std.TestMode THEN
		weight1 := DINT_TO_UINT(ABS(WeightRaw[1301].Wgt_Channel_1)/100);
		weight2 := DINT_TO_UINT(ABS(WeightRaw[1302].Wgt_Channel_1)/100);
		weight3 := DINT_TO_UINT(ABS(WeightRaw[1303].Wgt_Channel_1)/100);
		weight4 := DINT_TO_UINT(ABS(WeightRaw[1304].Wgt_Channel_1)/100);
		weight5 := DINT_TO_UINT(ABS(WeightRaw[1305].Wgt_Channel_1)/100);
		weight6 := DINT_TO_UINT(ABS(WeightRaw[1306].Wgt_Channel_1)/100);
		weight7 := DINT_TO_UINT(ABS(WeightRaw[1307].Wgt_Channel_1)/100);
		weight8 := DINT_TO_UINT(ABS(WeightRaw[1308].Wgt_Channel_1)/100);
		weight9 := DINT_TO_UINT(ABS(WeightRaw[1309].Wgt_Channel_1)/100);
		weight10 := DINT_TO_UINT(ABS(WeightRaw[1310].Wgt_Channel_1)/100);
		weight11 := DINT_TO_UINT(ABS(WeightRaw[1311].Wgt_Channel_1)/100);
		weight12 := DINT_TO_UINT(ABS(WeightRaw[1312].Wgt_Channel_1)/100);
		weight13 := DINT_TO_UINT(ABS(WeightRaw[1313].Wgt_Channel_1)/100);
		weight14 := DINT_TO_UINT(ABS(WeightRaw[1314].Wgt_Channel_1)/100);
		weight15 := DINT_TO_UINT(ABS(WeightRaw[1315].Wgt_Channel_1)/100);
		weight16 := DINT_TO_UINT(ABS(WeightRaw[1316].Wgt_Channel_1)/100);
		weight17 := DINT_TO_UINT(ABS(WeightRaw[1317].Wgt_Channel_1)/100);
		weight18 := DINT_TO_UINT(ABS(WeightRaw[1318].Wgt_Channel_1)/100);
	ELSE
		weight1 := testweight;
		weight2 := testweight;
		weight3 := testweight;
		weight4 := testweight;
		weight5 := testweight;
		weight6 := testweight;
		weight7 := testweight;
		weight8 := testweight;
		weight9 := testweight;
		weight10 := testweight;
		weight11 := testweight;
		weight12 := testweight;
		weight13 := testweight;
		weight14 := testweight;
		weight15 := testweight;
		weight16 := testweight;
		weight17 := testweight;
		weight18 := testweight;
	END_IF;

	//	weight19 := DINT_TO_UINT(ABS(WeightRaw[1319].Wgt_Channel_1)/100);
	//	weight20 := DINT_TO_UINT(ABS(WeightRaw[1320].Wgt_Channel_1)/100);
	//	weight21 := DINT_TO_UINT(ABS(WeightRaw[1321].Wgt_Channel_1)/100);
	//	weight22 := DINT_TO_UINT(ABS(WeightRaw[1322].Wgt_Channel_1)/100);
	//	weight23 := DINT_TO_UINT(ABS(WeightRaw[1323].Wgt_Channel_1)/100);
	//	weight24 := DINT_TO_UINT(ABS(WeightRaw[1324].Wgt_Channel_1)/100);
	//
	//	//Loading Units
	//	weight31 := DINT_TO_UINT(ABS(WeightRaw[1025].Wgt_Channel_1 + WeightRaw[1025].Wgt_Channel_2)/100); //SLU3
	//	weight32 := DINT_TO_UINT(ABS(WeightRaw[1027].Wgt_Channel_1 + WeightRaw[1027].Wgt_Channel_2)/100); //SLU4
	//	weight33 := DINT_TO_UINT(ABS(WeightRaw[1029].Wgt_Channel_1 + WeightRaw[1029].Wgt_Channel_2)/100); //SLU5
	//	weight34 := DINT_TO_UINT(ABS(WeightRaw[1621].Wgt_Channel_1 + WeightRaw[1621].Wgt_Channel_2)/100); //SLU6
	//
	//	//Weigh Beams
	//	weight48 := DINT_TO_UINT(ABS(WeightRaw[1339].Wgt_Channel_1)/100); //SWB1 ????
	//	weight49 := DINT_TO_UINT(ABS(WeightRaw[1340].Wgt_Channel_1)/100); //SWB2 ????

END_PROGRAM
```

### Sorting.var
```iecst
VAR CONSTANT
	MAX_STATIONS : USINT := 120; (*Maximum counting stations*)
	LIVE_DATA_TYPE_STATION_COUNTS : UINT := 5001; (*Packet ID for the UDP Packet*)
END_VAR
VAR
	SortingBins : Sorting_typ;
END_VAR
```

### Sorting.typ
```iecst
TYPE
	SortingItem_typ : 	STRUCT
		station : UINT;
		count : UINT;
		weight : UINT;
		cus : STRING[11];
		cat : STRING[11];
		spare1 : UINT;
		spare2 : UINT;
	END_STRUCT;
	Sorting_typ : 	STRUCT
		counting_frames : ARRAY[0..MAX_STATIONS]OF SortingItem_typ;
	END_STRUCT;
END_TYPE
```

### Program Logical/SortingSpecial/udpComm_disp (IEC, version 2.00.1) - udpComm

#### Main.st - Init, cyclic, exit code
```iecst
(*
----------------------------------------------------------------------------------------------------------------------------------------
--LIVE DATA TASK--
UDP MAX FRAME SIZE IS 65507 Bytes
-----------------------------------------------------------------------------------------------------------------------------------------
*)
//V1.00.1 -- 06/09/2019 -- First Version
//V1.00.2 -- 05/01/2020 -- Clean up basic version + Add dynamic start up for ABB drive data
//V2.00.1 -- 11/03/2020 -- Add Structures to replace TCP/IP Driver
PROGRAM _INIT
//Configure a static connection (Testing)
LiveDataConnection[1].Config.ServerIP 		:= '10.8.15.118'; //eVueServerIP;
LiveDataConnection[1].Config.ServerPort		:= 54321;
LiveDataConnection[1].Config.Type 			:= LIVE_DATA_CONFIG_STATIC;
//Create a fix request pool for test
LiveDataConnection[1].RequestPool.PoolList[1] 	:= LIVE_DATA_TYPE_STATION_COUNTS;

LiveDataConnection[1].RequestPool.PoolListSize 	:= 1;

//	SortingBins.counting_frames[1].station := 1;
//	SortingBins.counting_frames[1].cus := 'cus01';
//	SortingBins.counting_frames[1].cat := 'cat01';
//	SortingBins.counting_frames[1].count := 55;
//	SortingBins.counting_frames[1].weight := 123;

//_initialiseComms;
END_PROGRAM

PROGRAM _CYCLIC

  IF EDGEPOS(udpIdent_Error) THEN
    udpCloseAllIdent := 0;
    n := 0;
  END_IF;
  IF udpIdent_Error THEN // We have too many ports open -- temp stop all clients and close all udp connections.

    CASE udpCloseAllIdent OF

    0://Get list off all open idents
      ioctl ACCESS ADR(udpIoctl_Error);
      ioctl.enable := 1;
      ioctl.ident := udpINVALID_IDENT;
      ioctl.ioctl := udpID_LIST_GET;
      ioctl.pData := ADR(identInfo.IdentsList[0]);
      ioctl.datalen := SIZEOF(identInfo.IdentsList);
      ioctl();
      IF (ioctl.status = ERR_OK) THEN
        udpCloseAllIdent := 1;
      ELSIF (ioctl.status <> ERR_FUB_BUSY) THEN

      END_IF;

    1://Close all open connections

      close ACCESS ADR(udpClose_Error);
      close.enable := (identInfo.IdentsList[n] > 0);
      close.ident := identInfo.IdentsList[n];
      close();
      IF (close.status = ERR_OK) OR ((close.status <> ERR_FUB_BUSY) AND (close.status <> ERR_FUB_ENABLE_FALSE)) THEN
        identInfo.IdentsList[n] := 0;
        IF (n < 199) THEN
          n := n + 1;
        ELSE
          udpCloseAllIdent := 2;
        END_IF;
      ELSIF (identInfo.IdentsList[n] = 0) THEN
        udpCloseAllIdent := 2;
      END_IF;

    2:// Reinint all connections
      FOR n := 1 TO LIVE_DATA_MAX_CONNECTIONS DO
        connection ACCESS ADR(LiveDataConnection[n]);
        connection.State := LIVE_DATA_INIT;
      END_FOR;
      udpIdent_Error := 0;
      udpCloseAllIdent := 0;
    END_CASE;

  ELSE //Run
    FOR n := 1 TO LIVE_DATA_MAX_CONNECTIONS DO
      connection ACCESS ADR(LiveDataConnection[n]);
      CASE connection.State  OF
        LIVE_DATA_INIT: //Every connection must be initialised with server IP and Port. This can be static or dynamic via http GET.
          CASE connection.Config.Type OF
            LIVE_DATA_CONFIG_STATIC:
              //Check the IP is valid
              IF connection.Config.ServerIP <> '' THEN //Don;t check Port as this could be 0
                connection.State := LIVE_DATA_WAIT;
              END_IF;
            LIVE_DATA_CONFIG_DYNAMIC_CLIENT:
              //Http request to load the Server details + current request pool
            LIVE_DATA_CONFIG_DYNAMIC_SERVER;
              //Wait for a request on the http server to start a connection.
          END_CASE;

        LIVE_DATA_WAIT:
          _AddRemoveFromPool;
          //Wait for the Request pool to be greater than 0
          IF (connection.RequestPool.PoolListSize > 0) THEN
            connection.State := LIVE_DATA_OPEN_CONNECTION;
          END_IF;

        LIVE_DATA_OPEN_CONNECTION:
          //Open connection to serverr
          open ACCESS ADR(connection.Functions.Open);
          open.enable 	:= 1;
          open.options	:= 0;
          open.pIfAddr 	:= 0;//
          open.port		:= 0;//
          open();
          IF (open.status = ERR_OK) THEN
            connection.State := LIVE_DATA_SETUP_CONNECTION_TOS;
          ELSIF (open.status <> ERR_FUB_BUSY) THEN
            connection.Error := open.status;
            connection.State := LIVE_DATA_ERROR; // Go directly to error as the connection has failed
          END_IF;

        LIVE_DATA_SETUP_CONNECTION_TOS://Configure the UDP
          //We must set
          //1) Type of service 	-- udpIP_TOS_SET -- udpIP_TOS_RELIABILITY
          //2) Time to live 		--
          //Optional Send Buffer	-- udpSO_SNDBUF_SET

          //				udpIP_TOS_LOWDELAY			16
          //				udpIP_TOS_THROUGHPUT		8
          //				udpIP_TOS_RELIABILITY		4
          //				udpIP_TOS_MINCOST			2

          ioctl ACCESS ADR(connection.Functions.Ioctl);
          ioctl.enable := 1;
          ioctl.ident := connection.Functions.Open.ident;
          ioctl.ioctl := udpIP_TOS_SET;
          ioctl.pData := ADR(connection.Config.TOS);
          ioctl.datalen := 4;
          ioctl();
          IF (ioctl.status = ERR_OK) THEN
            connection.State := LIVE_DATA_SETUP_CONNECTION_TTL;
          ELSIF (ioctl.status <> ERR_FUB_BUSY) THEN
            connection.Error := ioctl.status;
            connection.State := LIVE_DATA_CLOSE_CONNECTION;
          END_IF;

        LIVE_DATA_SETUP_CONNECTION_TTL: //Time to LIVE in seconds -- MAX 255

          ioctl ACCESS ADR(connection.Functions.Ioctl);
          ioctl.enable := 1;
          ioctl.ident := connection.Functions.Open.ident;
          ioctl.ioctl := udpIP_TTL_SET;
          ioctl.pData := ADR(connection.Config.TTL);
          ioctl.datalen := 4;
          ioctl();
          IF (ioctl.status = ERR_OK) THEN
            connection.State := LIVE_DATA_CONNECT;
          ELSIF (ioctl.status <> ERR_FUB_BUSY) THEN
            connection.Error := ioctl.status;
            connection.State := LIVE_DATA_CLOSE_CONNECTION;
          END_IF;

        LIVE_DATA_CONNECT: // Connect to a specific Device (this is optional but improves performance)
          connect	ACCESS ADR(connection.Functions.Connect);
          connect.enable 	:= 1;
          connect.ident 	:= connection.Functions.Open.ident;
          connect.pHost	:= ADR(connection.Config.ServerIP);
          connect.port 	:= connection.Config.ServerPort;
          connect();
          IF (connect.status = ERR_OK) THEN
            IF getIdentInfo THEN
              connection.State := LIVE_DATA_GET_IDENT_LIST;
            ELSE
              connection.State := LIVE_DATA_BUILD_DATA;
            END_IF;
          ELSIF (connect.status <> ERR_FUB_BUSY) THEN
            connection.Error := connect.status;
            connection.State := LIVE_DATA_DISCONNECT;
          END_IF;
        LIVE_DATA_BUILD_DATA:
          //Build data-- Build a header and data combined.
          //Byte 1 		-- Request Type USINT
          //Byte 2 & 3	-- Header Size(Bytes) UINT
          //Byte 4,5,6,7	-- CheckSum		UDINT
          //Byte xxx		-- HEADER INFO -- BESPOKE TO Request Type
          //DATA--
          IF (connection.RequestPool.Pointer > 0) THEN
            CASE connection.RequestPool.PoolList[connection.RequestPool.Pointer] OF

//                LIVE_DATA_TYPE_DISP_UDP_COMM_1..LIVE_DATA_TYPE_DISP_UDP_COMM_5:
//                  //Built the packet
//                  udpComm[0] := connection.RequestPool.Pointer;
//                  FOR n := 1 TO DISP_SEND_PACKET_SIZE DO
//                    pointer :=  n + (DISP_SEND_PACKET_SIZE * (udpComm[0] - 1));
//                    IF (CommArrayDisp[pointer] <> 0) AND (pointer <= DISP_COMM_BUFFER_SIZE) THEN
//                      brsmemcpy(ADR(udpComm[n]),CommArrayDisp[pointer],2);
//                    ELSE
//                      udpComm[n] := 0;
//                    END_IF;
//                  END_FOR;
//                  pData := ADR(udpComm);
//                  length := SIZEOF(udpComm);
//                  connection.State := LIVE_DATA_SEND_DATA;
//
//                LIVE_DATA_TYPE_RAIL_MESSAGES:// Rail messages
//                  messages[0] := LIVE_DATA_TYPE_RAIL_MESSAGES;
//                  FOR n := 1 TO RAIL_COUNT DO
//                    messages[n] := RailComm[n].Messages.Write;
//                  END_FOR;
//                  pData := ADR(messages);
//                  length := SIZEOF(messages);
//                  connection.State := LIVE_DATA_SEND_DATA;
//
//                LIVE_DATA_TYPE_SLING_INPUT_STATE:// Sling input screen states.
//                  values[0] := LIVE_DATA_TYPE_SLING_INPUT_STATE;
//                  FOR n := 1 TO SLING_INPUTS_COUNT DO
//                    values[n] := SlingInputComm[n].Write;
//                  END_FOR;
//                  pData := ADR(values);
//                  length := ((SLING_INPUTS_COUNT + 1) * 2);
//                  connection.State := LIVE_DATA_SEND_DATA;

									LIVE_DATA_TYPE_STATION_COUNTS:
										values[0] := LIVE_DATA_TYPE_STATION_COUNTS;
										values[1] := MAX_STATIONS;

										length := SIZEOF(SortingBins);
										brsmemcpy(ADR(values[2]),ADR(SortingBins),length);
										length := length + 2;
										pData := ADR(values);
										connection.State := LIVE_DATA_SEND_DATA;

              ELSE
                //Invalid type- Check the pool again
                connection.State := LIVE_DATA_CHECK_REQUESTPOOL;
            END_CASE;
          ELSE
            connection.State := LIVE_DATA_CHECK_REQUESTPOOL;
          END_IF;

        LIVE_DATA_SEND_DATA:
          send ACCESS ADR(connection.Functions.Send);
          send.enable 	:= 1;
          send.ident 		:= connection.Functions.Open.ident;
          send.flags 		:= udpMSG_DONTROUTE;// Do not send via the gateway- Route Directly to Server
          send.pData 		:= pData;
          send.datalen	:= length;
          send();
          IF (send.status = ERR_OK) THEN
            connection.State := LIVE_DATA_CHECK_REQUESTPOOL;
          ELSIF send.status = udpERR_CONNREFUSED THEN // Server is not there, disconnect and start again
            connection.State := LIVE_DATA_DISCONNECT;
          ELSIF (send.status <> ERR_FUB_BUSY) THEN
            connection.Error := send.status;
            connection.State := LIVE_DATA_DISCONNECT;
          END_IF;

          //send.pHost || THESE ARE IGNORED BECAUSE WE ARE MAKING A DIRECT CONNECTION USING THE CONNECT FUB||
          //send.port

        LIVE_DATA_CHECK_REQUESTPOOL:
          //Check that the request pool hasn;t changed- Shuffle to the next Requested packet.
          _AddRemoveFromPool;
          //IF the pool is empty close the connection and wait
          IF (connection.RequestPool.Pointer = 0) AND (connection.RequestPool.PoolListSize > 0) THEN
            connection.RequestPool.Pointer := 1;
          ELSIF (connection.RequestPool.Pointer = connection.RequestPool.PoolListSize) THEN
            connection.RequestPool.Pointer := 1;
          ELSIF (connection.RequestPool.Pointer < connection.RequestPool.PoolListSize) THEN
            connection.RequestPool.Pointer := connection.RequestPool.Pointer + 1;
          ELSIF (connection.RequestPool.Pointer > connection.RequestPool.PoolListSize) AND (connection.RequestPool.PoolListSize > 0) THEN
            connection.RequestPool.Pointer := 1;
          END_IF;

          validConnection := (connection.Config.ServerIP <> '');
          IF (connection.RequestPool.PoolListSize = 0) OR NOT validConnection THEN
            connection.State := LIVE_DATA_DISCONNECT;
          ELSE
            connection.State := LIVE_DATA_BUILD_DATA;
          END_IF;

        LIVE_DATA_DISCONNECT:
          disconnect ACCESS ADR(connection.Functions.Disconnect);
          disconnect.enable := 1;
          disconnect.ident := connection.Functions.Open.ident;
          disconnect();
          IF (disconnect.status = ERR_OK) THEN
            connection.State := LIVE_DATA_CLOSE_CONNECTION;
          ELSIF (disconnect.status <> ERR_FUB_BUSY) THEN
            connection.Error := disconnect.status;
            connection.State := LIVE_DATA_CLOSE_CONNECTION;
          END_IF;

        LIVE_DATA_CLOSE_CONNECTION:
          close ACCESS ADR(connection.Functions.Close);
          close.enable := 1;
          close.ident := connection.Functions.Open.ident;
          close();
          IF (close.status = ERR_OK) THEN
            IF (connection.Error > 0) THEN
              connection.State := LIVE_DATA_ERROR;
            ELSE
              connection.State := LIVE_DATA_INIT;
            END_IF;
            IF (connection.Config.Type <> LIVE_DATA_CONFIG_STATIC) THEN
              connection.RequestPool 			:= CLEAR_REQUEST_POOL;
              connection.Config.ServerIP 		:= '';
              connection.Config.ServerPort 	:= 0;
            END_IF;

          ELSIF (close.status <> ERR_FUB_BUSY) THEN
            connection.Error := close.status ;
            connection.State := LIVE_DATA_ERROR;
          END_IF;

        LIVE_DATA_ERROR:
          IF (connection.Error = udpERR_NOMORE_IDENTS) THEN
            // All Idents are used we have to close them manually.
            udpIdent_Error := 1;
          ELSE
            errorCount := errorCount + 1;
            connection.Error := 0;
            connection.State := LIVE_DATA_INIT;
          END_IF;

        LIVE_DATA_GET_IDENT_LIST:
          ioctl ACCESS ADR(connection.Functions.Ioctl);
          ioctl.enable := 1;
          ioctl.ident := udpINVALID_IDENT;
          ioctl.ioctl := udpID_LIST_GET;
          ioctl.pData := ADR(identInfo.IdentsList[0]);
          ioctl.datalen := SIZEOF(identInfo.IdentsList);
          ioctl();
          IF (ioctl.status = ERR_OK) THEN
            connection.State := LIVE_DATA_GET_IDENT_MAX;
          ELSIF (ioctl.status <> ERR_FUB_BUSY) THEN

          END_IF;

        LIVE_DATA_GET_IDENT_MAX:
          ioctl ACCESS ADR(connection.Functions.Ioctl);
          ioctl.enable := 1;
          ioctl.ident := udpINVALID_IDENT;
          ioctl.ioctl := udpID_MAX_GET;
          ioctl.pData := ADR(identInfo.MaxIdents);
          ioctl.datalen := 4;
          ioctl();
          IF (ioctl.status = ERR_OK) THEN
            connection.State := LIVE_DATA_BUILD_DATA;
          ELSIF (ioctl.status <> ERR_FUB_BUSY) THEN

          END_IF;

      END_CASE;

    END_FOR;
  END_IF;

END_PROGRAM

PROGRAM _EXIT
  // DO we have to close the connections on EXIT -- Perhaps when a transfer happens!!

END_PROGRAM
```

#### _initialiseComms.st
```iecst
// Initialise the Comm registers.
ACTION _initialiseComms:
  //Generated Init Code.
//	FOR n := 0 TO DISP_COMM_BUFFER_SIZE DO
//		CommArrayDisp[n] := 0;
//	END_FOR;
//
//	FOR n := 1 TO MAX_STATIONS DO
//		CommArrayDisp[n] := ADR(SortingBins.counting_frames[n]);
//	END_FOR;

END_ACTION
```

#### Types.typ - Local data types
```iecst
TYPE
	identInfo_typ : 	STRUCT
		MaxIdents : UDINT;
		IdentsList : ARRAY[0..199]OF UDINT;
	END_STRUCT;
END_TYPE
```

#### Variables.var - Local variables
```iecst
VAR CONSTANT
	CLEAR_REQUEST_POOL : LiveData_RequestPool_typ := (AddToPool:=0,RemoveFromPool:=0,PoolListSize:=0,Pointer:=0);
END_VAR
VAR
	n : UINT;
	pointer : UDINT;
	connection : REFERENCE TO LiveDataConnection_typ;
	LiveDataConnection : ARRAY[1..LIVE_DATA_MAX_CONNECTIONS] OF LiveDataConnection_typ;
	udpComm : ARRAY[0..UDP_SEND_PACKET_SIZE] OF UINT;
	open : REFERENCE TO UdpOpen;
	ioctl : REFERENCE TO UdpIoctl;
	connect : REFERENCE TO UdpConnect;
	send : REFERENCE TO UdpSend;
	pData : UDINT;
	length : UDINT;
	disconnect : REFERENCE TO UdpDisconnect;
	close : REFERENCE TO UdpClose;
	errorCount : UDINT;
	validConnection : BOOL;
	i : USINT;
	identInfo : identInfo_typ;
	getIdentInfo : BOOL;
	udpIdent_Error : BOOL;
	udpIoctl_Error : UdpIoctl;
	udpCloseAllIdent : USINT;
	udpClose_Error : UdpClose;
	data : ARRAY[0..65534] OF SINT; (**Max data frame that can be sent by UDP*)
	values : ARRAY[0..2000] OF UINT;
END_VAR
```

### Global _backup.var - not listed in the package file held
```iecst
VAR
	X : ARRAY[0..1400] OF bnr_io;
	Y : ARRAY[0..1400] OF bnr_io;
	OK : ARRAY[0..1400] OF BOOL;
	StnOK : ARRAY[0..1400] OF BOOL;
	spare : BOOL;
	SPARE : BOOL;
	spare_input : BOOL;
	r6_route_sensor : BOOL;
	r6_align_in_sensor_b : BOOL;
	r6_align_in_sensor_a : BOOL;
	r6_align_out_sensor_a : BOOL;
	r6_align_out_sensor_b : BOOL;
	r6_rotate_in : BOOL;
	r6_safety_stop : BOOL;
	r6_rotate_out : BOOL;
	lift_safety_10 : BOOL;
	lift_safety_11 : BOOL;
	lift_safety_12 : BOOL;
	lift_safety_18 : BOOL;
	spare_output : BOOL;
	unknown_input : BOOL;
	unknown_output : BOOL;
	plc_info1 : WORD;
	plc_info2 : WORD;
	ss1 : BOOL;
	ss2 : BOOL;
	ss3 : BOOL;
	ss4 : BOOL;
	ss5 : BOOL;
	ss6 : BOOL;
	ss7 : BOOL;
	ss8 : BOOL;
	ss9 : BOOL;
	ss10 : BOOL;
	ss1_prs : BOOL;
	ss2_prs : BOOL;
	ss3_prs : BOOL;
	ss4_prs : BOOL;
	ss5_prs : BOOL;
	ss6_prs : BOOL;
	ss7_prs : BOOL;
	ss8_prs : BOOL;
	ss9_prs : BOOL;
	ss10_prs : BOOL;
	r1 : rail;
	r1_R_TRIG1 : R_TRIG;
	r1_R_TRIG2 : R_TRIG;
	r1_R_TRIG3 : R_TRIG;
	r1_R_TRIG4 : R_TRIG;
	r1_R_TRIG5 : R_TRIG;
	r1_R_TRIG6 : R_TRIG;
	r1_R_TRIG7 : R_TRIG;
	r1_R_TRIG8 : R_TRIG;
	r1_R_TRIG9 : R_TRIG;
	r1_R_TRIG10 : R_TRIG;
	r1_R_TRIG11 : R_TRIG;
	r1_F_TRIG1 : F_TRIG;
	r1_F_TRIG2 : F_TRIG;
	r1_F_TRIG3 : F_TRIG;
	r1_F_TRIG4 : F_TRIG;
	r1_ALM : TON;
	r1_WARN : TON;
	r2 : rail;
	r2_R_TRIG1 : R_TRIG;
	r2_R_TRIG2 : R_TRIG;
	r2_R_TRIG3 : R_TRIG;
	r2_R_TRIG4 : R_TRIG;
	r2_R_TRIG5 : R_TRIG;
	r2_R_TRIG6 : R_TRIG;
	r2_R_TRIG7 : R_TRIG;
	r2_R_TRIG8 : R_TRIG;
	r2_R_TRIG9 : R_TRIG;
	r2_R_TRIG10 : R_TRIG;
	r2_R_TRIG11 : R_TRIG;
	r2_F_TRIG1 : F_TRIG;
	r2_F_TRIG2 : F_TRIG;
	r2_F_TRIG3 : F_TRIG;
	r2_F_TRIG4 : F_TRIG;
	r2_ALM : TON;
	r2_WARN : TON;
	r3 : rail;
	r3_ALM : TON;
	r3_WARN : TON;
	r4 : rail;
	r4_XFR_R_TRIG1 : R_TRIG;
	r4_XFR_R_TRIG2 : R_TRIG;
	r4_SW_R_TRIG1 : R_TRIG;
	r4_SW_R_TRIG2 : R_TRIG;
	r4_ALM : TON;
	r4_WARN : TON;
	r5 : rail;
	r5_ALM : TON;
	r5_WARN : TON;
	r6 : rail;
	r6_SW_R_TRIG1 : R_TRIG;
	r6_SW_R_TRIG2 : R_TRIG;
	r6_ALM : TON;
	r6_WARN : TON;
	r7 : rail;
	r7_ALM : TON;
	r7_WARN : TON;
	r8 : rail;
	r8_R_TRIG1 : R_TRIG;
	r8_R_TRIG2 : R_TRIG;
	r8_ALM : TON;
	r8_WARN : TON;
	r9 : rail;
	r9_ALM : TON;
	r9_WARN : TON;
	r10 : rail;
	r10_ALM : TON;
	r10_WARN : TON;
	r11 : rail;
	r11_ALM : TON;
	r11_WARN : TON;
	r12 : rail;
	r12_ALM : TON;
	r12_WARN : TON;
	r13 : rail;
	r13_ALM : TON;
	r13_WARN : TON;
	r14 : rail;
	r14_R_TRIG1 : R_TRIG;
	r14_R_TRIG2 : R_TRIG;
	r14_R_TRIG3 : R_TRIG;
	r14_F_TRIG1 : F_TRIG;
	r14_ALM : TON;
	r14_WARN : TON;
	r15 : rail;
	r15_ALM : TON;
	r15_WARN : TON;
	r16 : rail;
	r16_R_TRIG1 : R_TRIG;
	r16_R_TRIG2 : R_TRIG;
	r16_R_TRIG3 : R_TRIG;
	r16_F_TRIG1 : F_TRIG;
	r16_ALM : TON;
	r16_WARN : TON;
	r17 : rail;
	r17_SW_R_TRIG1 : R_TRIG;
	r17_SW_R_TRIG2 : R_TRIG;
	r17_ALM : TON;
	r17_WARN : TON;
	r18 : rail;
	r18_SW_R_TRIG1 : R_TRIG;
	r18_SW_R_TRIG2 : R_TRIG;
	r18_ALM : TON;
	r18_WARN : TON;
	r19 : rail;
	r19_R_TRIG1 : R_TRIG;
	r19_R_TRIG2 : R_TRIG;
	r19_R_TRIG3 : R_TRIG;
	r19_F_TRIG1 : F_TRIG;
	r19_ALM : TON;
	r19_WARN : TON;
	r20 : rail;
	r20_R_TRIG1 : R_TRIG;
	r20_R_TRIG2 : R_TRIG;
	r20_SW_R_TRIG1 : R_TRIG;
	r20_SW_R_TRIG2 : R_TRIG;
	r20_ALM : TON;
	r20_WARN : TON;
	r21 : rail;
	r21_R_TRIG1 : R_TRIG;
	r21_R_TRIG2 : R_TRIG;
	r21_SW_R_TRIG1 : R_TRIG;
	r21_SW_R_TRIG2 : R_TRIG;
	r21_ALM : TON;
	r21_WARN : TON;
	r22 : rail;
	r22_ALM : TON;
	r22_WARN : TON;
	one_sec_pulse : TON;
	not_one_sec_pulse : TON;
	thirty_msec_pulse : TON;
	not_thirty_msec_pulse : TON;
	conveyor_module_1_value_1 : INT;
	conveyor_module_1_value_2 : INT;
	conveyor_module_1_value_3 : INT;
	conveyor_module_1_value_4 : INT;
	conveyor_module_2_value_1 : INT;
	conveyor_module_2_value_2 : INT;
	conveyor_module_2_value_3 : INT;
	conveyor_module_2_value_4 : INT;
	conveyor_module_3_value_1 : INT;
	conveyor_module_3_value_2 : INT;
	conveyor_module_3_value_3 : INT;
	conveyor_module_3_value_4 : INT;
	conveyor_module_4_value_1 : INT;
	conveyor_module_4_value_2 : INT;
	conveyor_module_4_value_3 : INT;
	conveyor_module_4_value_4 : INT;
	conveyor_module_5_value_1 : INT;
	conveyor_module_5_value_2 : INT;
	conveyor_module_5_value_3 : INT;
	conveyor_module_5_value_4 : INT;
	conveyor_module_6_value_1 : INT;
	conveyor_module_6_value_2 : INT;
	conveyor_module_6_value_3 : INT;
	conveyor_module_6_value_4 : INT;
	conveyor_module_7_value_1 : INT;
	conveyor_module_7_value_2 : INT;
	conveyor_module_7_value_3 : INT;
	conveyor_module_7_value_4 : INT;
	conveyor_module_8_value_1 : INT;
	conveyor_module_8_value_2 : INT;
	conveyor_module_8_value_3 : INT;
	conveyor_module_8_value_4 : INT;
	conveyor_module_9_value_1 : INT;
	conveyor_module_9_value_2 : INT;
	conveyor_module_9_value_3 : INT;
	conveyor_module_9_value_4 : INT;
	conveyor_module_10_value_1 : INT;
	conveyor_module_10_value_2 : INT;
	conveyor_module_10_value_3 : INT;
	conveyor_module_10_value_4 : INT;
	conveyor_module_11_value_1 : INT;
	conveyor_module_11_value_2 : INT;
	conveyor_module_11_value_3 : INT;
	conveyor_module_11_value_4 : INT;
	conveyor_module_12_value_1 : INT;
	conveyor_module_12_value_2 : INT;
	conveyor_module_12_value_3 : INT;
	conveyor_module_12_value_4 : INT;
	conveyor_module_13_value_1 : INT;
	conveyor_module_13_value_2 : INT;
	conveyor_module_13_value_3 : INT;
	conveyor_module_13_value_4 : INT;
	conveyor_module_14_value_1 : INT;
	conveyor_module_14_value_2 : INT;
	conveyor_module_14_value_3 : INT;
	conveyor_module_14_value_4 : INT;
	conveyor_module_15_value_1 : INT;
	conveyor_module_15_value_2 : INT;
	conveyor_module_15_value_3 : INT;
	conveyor_module_15_value_4 : INT;
	conveyor_module_16_value_1 : INT;
	conveyor_module_16_value_2 : INT;
	conveyor_module_16_value_3 : INT;
	conveyor_module_16_value_4 : INT;
	conveyor_module_17_value_1 : INT;
	conveyor_module_17_value_2 : INT;
	conveyor_module_17_value_3 : INT;
	conveyor_module_17_value_4 : INT;
	conveyor_module_18_value_1 : INT;
	conveyor_module_18_value_2 : INT;
	conveyor_module_18_value_3 : INT;
	conveyor_module_18_value_4 : INT;
	conveyor_module_19_value_1 : INT;
	conveyor_module_19_value_2 : INT;
	conveyor_module_19_value_3 : INT;
	conveyor_module_19_value_4 : INT;
	ModbusTcpMaster_Array : ARRAY[0..23] OF MBmaster;
	MasterConfig_Array : ARRAY[0..23] OF modbus_master_cfg_typ;
	ip : STRING[80];
	StartStop : BOOL;
	WeightRaw : ARRAY[1..1001] OF Weight_typ;
	weight1a : DINT;
	weight1b : DINT;
	weight1c : DINT;
	weight1d : DINT;
	weight2a : DINT;
	weight2b : DINT;
	weight2c : DINT;
	weight2d : DINT;
	Weights : ARRAY[0..2] OF UINT;
	myRaw1 : DINT;
	myRaw2 : DINT;
	r4_tran_ON1 : TON;
	r4_tran_F_TRIG1 : F_TRIG;
	b1_xfr_ok : BOOL;
	b1_srt_1 : TON;
	b1_x_complete : BOOL;
	b1_conv_ok : BOOL;
	b1_conv : BOOL;
	r3_wrn_off : TOF;
	run_conveyor_1_fwd : BOOL;
	r10_fire : BOOL;
	r11_fire : BOOL;
	r13_fire : BOOL;
	r16_clamp : BOOL;
	r16_rail_in_prs : BOOL;
	r16_rail_out_prs : BOOL;
	r16_move_rail_in : BOOL;
	r10_position : USINT;
	r11_position : USINT;
	r13_position : USINT;
	r9_wrn_off : TOF;
	r9_TON1 : TON;
	r9_TON2 : TON;
	r9_TON3 : TON;
	r9_TON4 : TON;
	r8_dump_send : BOOL;
	r16_clamp_off : TOF;
END_VAR
VAR RETAIN
	validation_alarm : BOOL;
	halted : BOOL;
	server_status : WORD;
	system_alarm_1 : BOOL;
	strobe1 : BOOL;
	horn1 : BOOL;
	system_alarm_2 : BOOL;
	strobe2 : BOOL;
	horn2 : BOOL;
	rail_alarm_time_1 : INT;
	rail_warning_1 : WORD;
	warn1 : BOOL;
	rail_signal_1 : WORD;
	rail_status_1 : WORD;
	r1_DBNC_arrive_OFF : TOF;
	r1_DBNC_before_OFF : TOF;
	r1_DBNC_after_OFF : TOF;
	r1_WRN1_ON : TON;
	r1_SRT1_ON : TON;
	r1_SRT2_ON : TON;
	r1_SRT3_OFF : TOF;
	rail_alarm_time_2 : INT;
	rail_warning_2 : WORD;
	warn2 : BOOL;
	rail_signal_2 : WORD;
	rail_status_2 : WORD;
	r2_DBNC_arrive_OFF : TOF;
	r2_DBNC_before_OFF : TOF;
	r2_DBNC_after_OFF : TOF;
	r2_WRN1_ON : TON;
	r2_SRT1_ON : TON;
	r2_SRT2_ON : TON;
	r2_SRT3_OFF : TOF;
	rail_alarm_time_3 : INT;
	rail_warning_3 : WORD;
	warn3 : BOOL;
	rail_signal_3 : WORD;
	rail_status_3 : WORD;
	r3_DBNC_front_ON : TON;
	r3_DBNC_arrive_ON : TON;
	r3_DBNC_after_OFF : TOF;
	r3_WRN1_ON : TON;
	rail_alarm_time_4 : INT;
	rail_warning_4 : WORD;
	warn4 : BOOL;
	rail_signal_4 : WORD;
	rail_status_4 : WORD;
	r4_DBNC_front_ON : TON;
	r4_DBNC_up_ON : TON;
	r4_DBNC_down_ON : TON;
	r4_DBNC_mid_ON : TON;
	r4_DBNC_arrive_ON : TON;
	r4_DBNC_before_OFF : TOF;
	r4_DBNC_after_OFF : TOF;
	r4_WRN1_ON : TON;
	r4_CB1_ON : TON;
	r4_CB2_ON : TON;
	rail_alarm_time_5 : INT;
	rail_warning_5 : WORD;
	warn5 : BOOL;
	rail_signal_5 : WORD;
	rail_status_5 : WORD;
	r5_DBNC_front_ON : TON;
	r5_DBNC_arrive_OFF : TOF;
	r5_DBNC_after_OFF : TOF;
	r5_WRN1_ON : TON;
	rail_alarm_time_6 : INT;
	rail_warning_6 : WORD;
	warn6 : BOOL;
	rail_signal_6 : WORD;
	rail_status_6 : WORD;
	r6_DBNC_front_ON : TON;
	r6_DBNC_arrive_OFF : TOF;
	r6_DBNC_after_OFF : TOF;
	r6_DBNC_before_OFF : TOF;
	rail_alarm_time_7 : INT;
	rail_warning_7 : WORD;
	warn7 : BOOL;
	rail_signal_7 : WORD;
	rail_status_7 : WORD;
	r7_DBNC_front_ON : TON;
	r7_DBNC_arrive_OFF : TOF;
	r7_DBNC_after_OFF : TOF;
	r7_WRN1_ON : TON;
	rail_alarm_time_8 : INT;
	rail_warning_8 : WORD;
	warn8 : BOOL;
	rail_signal_8 : WORD;
	rail_status_8 : WORD;
	r8_DBNC_front_ON : TON;
	r8_DBNC_arrive_ON : TON;
	r8_DBNC_after_OFF : TOF;
	r8_OPN1_ON : TON;
	r8_OPN2_ON : TON;
	r8_OPN5_ON : TON;
	r8_OPN6_ON : TON;
	r8_OPN7_ON : TON;
	r8_OPN8_ON : TON;
	r8_OPN9_ON : TON;
	r8_WRN1_ON : TON;
	r8_OPN3_OFF : TOF;
	r8_OPN4_OFF : TOF;
	rail_alarm_time_9 : INT;
	rail_warning_9 : WORD;
	warn9 : BOOL;
	rail_signal_9 : WORD;
	rail_status_9 : WORD;
	r9_DBNC_front_ON : TON;
	r9_DBNC_arrive_OFF : TOF;
	rail_alarm_time_10 : INT;
	rail_warning_10 : WORD;
	warn10 : BOOL;
	rail_signal_10 : WORD;
	rail_status_10 : WORD;
	r10_DBNC_front_ON : TON;
	r10_DBNC_arrive_OFF : TOF;
	r10_DBNC_after_OFF : TOF;
	r10_WRN1_ON : TON;
	rail_alarm_time_11 : INT;
	rail_warning_11 : WORD;
	warn11 : BOOL;
	rail_signal_11 : WORD;
	rail_status_11 : WORD;
	r11_DBNC_front_ON : TON;
	r11_DBNC_arrive_OFF : TOF;
	r11_DBNC_after_OFF : TOF;
	r11_WRN1_ON : TON;
	rail_alarm_time_12 : INT;
	rail_warning_12 : WORD;
	warn12 : BOOL;
	rail_signal_12 : WORD;
	rail_status_12 : WORD;
	r12_DBNC_front_ON : TON;
	r12_DBNC_arrive_OFF : TOF;
	r12_DBNC_after_OFF : TOF;
	r12_WRN1_ON : TON;
	rail_alarm_time_13 : INT;
	rail_warning_13 : WORD;
	warn13 : BOOL;
	rail_signal_13 : WORD;
	rail_status_13 : WORD;
	r13_DBNC_front_ON : TON;
	r13_DBNC_arrive_ON : TON;
	r13_DBNC_after_OFF : TOF;
	r13_WRN1_ON : TON;
	rail_alarm_time_14 : INT;
	rail_warning_14 : WORD;
	warn14 : BOOL;
	rail_signal_14 : WORD;
	rail_status_14 : WORD;
	r14_DBNC_front_ON : TON;
	r14_DBNC_arrive_ON : TON;
	r14_DBNC_up_ON : TON;
	r14_DBNC_down_ON : TON;
	r14_DBNC_after_OFF : TOF;
	r14_WRN1_ON : TON;
	rail_alarm_time_15 : INT;
	rail_warning_15 : WORD;
	warn15 : BOOL;
	rail_signal_15 : WORD;
	rail_status_15 : WORD;
	r15_DBNC_front_ON : TON;
	r15_DBNC_arrive_ON : TON;
	r15_DBNC_after_OFF : TOF;
	r15_WRN1_ON : TON;
	rail_alarm_time_16 : INT;
	rail_warning_16 : WORD;
	warn16 : BOOL;
	rail_signal_16 : WORD;
	rail_status_16 : WORD;
	r16_DBNC_front_ON : TON;
	r16_DBNC_up_ON : TON;
	r16_DBNC_arrive_OFF : TOF;
	r16_DBNC_after_OFF : TOF;
	r16_LFT1_ON : TON;
	r16_LFT2_ON : TON;
	r16_LFT3_ON : TON;
	r16_LFT5_ON : TON;
	r16_WRN1_ON : TON;
	r16_LFT4_OFF : TOF;
	rail_alarm_time_17 : INT;
	rail_warning_17 : WORD;
	warn17 : BOOL;
	rail_signal_17 : WORD;
	rail_status_17 : WORD;
	r17_DBNC_front_ON : TON;
	r17_DBNC_arrive_OFF : TOF;
	r17_DBNC_after_OFF : TOF;
	r17_DBNC_before_OFF : TOF;
	rail_alarm_time_18 : INT;
	rail_warning_18 : WORD;
	warn18 : BOOL;
	rail_signal_18 : WORD;
	rail_status_18 : WORD;
	r18_DBNC_front_ON : TON;
	r18_DBNC_arrive_OFF : TOF;
	r18_DBNC_after_OFF : TOF;
	r18_DBNC_before_OFF : TOF;
	rail_alarm_time_19 : INT;
	rail_warning_19 : WORD;
	warn19 : BOOL;
	rail_signal_19 : WORD;
	rail_status_19 : WORD;
	r19_DBNC_arrive_OFF : TOF;
	r19_DBNC_after_OFF : TOF;
	r19_WRN1_ON : TON;
	rail_alarm_time_20 : INT;
	rail_warning_20 : WORD;
	warn20 : BOOL;
	rail_signal_20 : WORD;
	rail_status_20 : WORD;
	r20_DBNC_front_ON : TON;
	r20_DBNC_arrive_ON : TON;
	r20_DBNC_after_OFF : TOF;
	r20_DBNC_before_OFF : TOF;
	r20_CLS1_ON : TON;
	r20_CLS3_ON : TON;
	r20_CLS2_OFF : TOF;
	r20_CLS4_OFF : TOF;
	rail_alarm_time_21 : INT;
	rail_warning_21 : WORD;
	warn21 : BOOL;
	rail_signal_21 : WORD;
	rail_status_21 : WORD;
	r21_DBNC_front_ON : TON;
	r21_DBNC_arrive_ON : TON;
	r21_DBNC_after_OFF : TOF;
	r21_DBNC_before_OFF : TOF;
	r21_CLS1_ON : TON;
	r21_CLS3_ON : TON;
	r21_CLS2_OFF : TOF;
	r21_CLS4_OFF : TOF;
	rail_alarm_time_22 : INT;
	rail_warning_22 : WORD;
	warn22 : BOOL;
	rail_signal_22 : WORD;
	rail_status_22 : WORD;
	r22_DBNC_front_ON : TON;
	r22_DBNC_arrive_ON : TON;
	r22_DBNC_after_OFF : TOF;
	r22_WRN1_ON : TON;
	sort_status_1 : WORD;
	sort_status_2 : WORD;
	M011_IN : ARRAY[0..40] OF INT;
	M011_OUT : ARRAY[0..40] OF INT;
	M012_IN : ARRAY[0..40] OF INT;
	M012_OUT : ARRAY[0..40] OF INT;
	M041_IN : ARRAY[0..40] OF INT;
	M041_OUT : ARRAY[0..40] OF INT;
	M051_IN : ARRAY[0..40] OF INT;
	M051_OUT : ARRAY[0..40] OF INT;
	M061_IN : ARRAY[0..40] OF INT;
	M061_OUT : ARRAY[0..40] OF INT;
	M081_IN : ARRAY[0..40] OF INT;
	M081_OUT : ARRAY[0..40] OF INT;
	M082_IN : ARRAY[0..40] OF INT;
	M082_OUT : ARRAY[0..40] OF INT;
	M091_IN : ARRAY[0..40] OF INT;
	M091_OUT : ARRAY[0..40] OF INT;
	M092_IN : ARRAY[0..40] OF INT;
	M092_OUT : ARRAY[0..40] OF INT;
	M101_IN : ARRAY[0..40] OF INT;
	M101_OUT : ARRAY[0..40] OF INT;
	M111_IN : ARRAY[0..40] OF INT;
	M111_OUT : ARRAY[0..40] OF INT;
	M112_IN : ARRAY[0..40] OF INT;
	M112_OUT : ARRAY[0..40] OF INT;
	M201_IN : ARRAY[0..40] OF INT;
	M201_OUT : ARRAY[0..40] OF INT;
	M301_IN : ARRAY[0..40] OF INT;
	M301_OUT : ARRAY[0..40] OF INT;
	M302_IN : ARRAY[0..40] OF INT;
	M302_OUT : ARRAY[0..40] OF INT;
	M303_IN : ARRAY[0..40] OF INT;
	M303_OUT : ARRAY[0..40] OF INT;
	M304_IN : ARRAY[0..40] OF INT;
	M304_OUT : ARRAY[0..40] OF INT;
	M401_IN : ARRAY[0..40] OF INT;
	M401_OUT : ARRAY[0..40] OF INT;
	M402_IN : ARRAY[0..40] OF INT;
	M402_OUT : ARRAY[0..40] OF INT;
	M403_IN : ARRAY[0..40] OF INT;
	M403_OUT : ARRAY[0..40] OF INT;
	M501_IN : ARRAY[0..40] OF INT;
	M501_OUT : ARRAY[0..40] OF INT;
	M502_IN : ARRAY[0..40] OF INT;
	M502_OUT : ARRAY[0..40] OF INT;
	M503_IN : ARRAY[0..40] OF INT;
	M503_OUT : ARRAY[0..40] OF INT;
	M1001_IN : ARRAY[0..40] OF INT;
	M1001_OUT : ARRAY[0..40] OF INT;
	PANEL_ONLINE_1 : INT;
	PANEL_ONLINE_2 : INT;
	weight1 : INT;
	capture_weight_1 : INT;
	min_weight_1 : INT;
	near_weight_1 : INT;
	buffer_weight_1 : INT;
	notify_weight_1 : INT;
	send_weight_1 : INT;
	over_weight_1 : INT;
	weight2 : INT;
	capture_weight_2 : INT;
	min_weight_2 : INT;
	near_weight_2 : INT;
	buffer_weight_2 : INT;
	notify_weight_2 : INT;
	send_weight_2 : INT;
	over_weight_2 : INT;
	force_enabled_comm_1 : WORD;
	force_value_comm_1 : WORD;
	io_comm_1 : WORD;
	force_enabled_comm_2 : WORD;
	force_value_comm_2 : WORD;
	io_comm_2 : WORD;
	force_enabled_comm_3 : WORD;
	force_value_comm_3 : WORD;
	io_comm_3 : WORD;
	force_enabled_comm_4 : WORD;
	force_value_comm_4 : WORD;
	io_comm_4 : WORD;
	force_enabled_comm_5 : WORD;
	force_value_comm_5 : WORD;
	io_comm_5 : WORD;
	force_enabled_comm_6 : WORD;
	force_value_comm_6 : WORD;
	io_comm_6 : WORD;
	force_enabled_comm_7 : WORD;
	force_value_comm_7 : WORD;
	io_comm_7 : WORD;
	force_enabled_comm_8 : WORD;
	force_value_comm_8 : WORD;
	io_comm_8 : WORD;
	force_enabled_comm_9 : WORD;
	force_value_comm_9 : WORD;
	io_comm_9 : WORD;
	force_enabled_comm_10 : WORD;
	force_value_comm_10 : WORD;
	io_comm_10 : WORD;
	force_enabled_comm_11 : WORD;
	force_value_comm_11 : WORD;
	io_comm_11 : WORD;
	insert_reset_1 : WORD;
	waiting_1 : WORD;
	insert_1 : WORD;
	bring_ok_1 : WORD;
	alarm_1 : WORD;
	insert_reset_2 : WORD;
	waiting_2 : WORD;
	insert_2 : WORD;
	bring_ok_2 : WORD;
	alarm_2 : WORD;
	rail_destination_1 : INT;
	rail_destination_2 : INT;
	rail_destination_3 : INT;
	rail_destination_4 : INT;
	rail_destination_5 : INT;
	rail_destination_6 : INT;
	rail_destination_7 : INT;
	rail_destination_8 : INT;
	rail_destination_9 : INT;
	rail_destination_10 : INT;
	rail_destination_11 : INT;
	rail_destination_12 : INT;
	rail_destination_13 : INT;
	rail_destination_14 : INT;
	rail_destination_15 : INT;
	rail_destination_16 : INT;
	rail_destination_17 : INT;
	rail_destination_18 : INT;
	rail_destination_19 : INT;
	rail_destination_20 : INT;
	rail_destination_21 : INT;
	rail_destination_22 : INT;
	rail_destination_23 : INT;
	rail_destination_24 : INT;
	rail_destination_25 : INT;
	rail_destination_26 : INT;
	rail_destination_27 : INT;
	rail_destination_28 : INT;
	rail_destination_29 : INT;
	rail_destination_30 : INT;
	rail_destination_31 : INT;
	rail_destination_32 : INT;
	rail_destination_33 : INT;
	rail_destination_34 : INT;
	rail_destination_35 : INT;
	rail_destination_36 : INT;
	rail_destination_37 : INT;
	rail_destination_38 : INT;
	rail_destination_39 : INT;
	rail_destination_40 : INT;
	rail_destination_41 : INT;
	rail_destination_42 : INT;
	rail_destination_43 : INT;
	rail_destination_44 : INT;
	rail_destination_45 : INT;
	rail_destination_46 : INT;
	rail_destination_47 : INT;
	rail_destination_48 : INT;
	rail_destination_49 : INT;
	rail_destination_50 : INT;
	rail_destination_51 : INT;
	rail_destination_52 : INT;
	rail_destination_53 : INT;
	rail_destination_54 : INT;
	rail_destination_55 : INT;
	rail_destination_56 : INT;
	rail_destination_57 : INT;
	rail_destination_58 : INT;
	rail_destination_59 : INT;
	rail_destination_60 : INT;
	rail_destination_61 : INT;
	rail_destination_62 : INT;
	rail_destination_63 : INT;
	rail_destination_64 : INT;
	rail_destination_65 : INT;
	rail_destination_66 : INT;
	rail_destination_67 : INT;
	rail_destination_68 : INT;
	rail_destination_69 : INT;
	rail_destination_70 : INT;
	rail_destination_71 : INT;
	rail_destination_72 : INT;
	rail_destination_73 : INT;
	rail_destination_74 : INT;
	rail_destination_75 : INT;
	rail_destination_76 : INT;
	rail_destination_77 : INT;
	rail_destination_78 : INT;
	rail_destination_79 : INT;
	rail_destination_80 : INT;
	rail_destination_81 : INT;
	rail_destination_82 : INT;
	rail_destination_83 : INT;
	rail_destination_84 : INT;
	rail_destination_85 : INT;
	rail_destination_86 : INT;
	rail_destination_87 : INT;
	rail_destination_88 : INT;
	rail_destination_89 : INT;
	rail_destination_90 : INT;
	rail_destination_91 : INT;
	rail_destination_92 : INT;
	rail_destination_93 : INT;
	rail_destination_94 : INT;
	rail_destination_95 : INT;
	rail_destination_96 : INT;
	rail_destination_97 : INT;
	rail_destination_98 : INT;
	rail_destination_99 : INT;
	rail_destination_100 : INT;
	rail_destination_101 : INT;
	DEST_SIZE : INT;
	DEST_NUM : INT;
	DEST_RAIL : INT;
	DEST_INDEX : INT;
END_VAR
```

Listed in the project but not available here: Logical/Standard/IOLink/Contactron/IOLink.var, Logical/Standard/IOLink/Contactron/Contactron/Types.typ, Logical/Standard/ToDO/Kanlink, Logical/Rails, Logical/COMMUNICATION/MbusTCP/MbusTCP.fun, Logical/COMMUNICATION/tcpComm/_initialiseComms.st, Logical/Safety/Safety/Types.typ, Logical/Safety/mappSafety/Types.typ, Logical/OPCuA_Client/OPCuAClient/Types.typ, Logical/http_Lib/KanHttp/Types.typ, Logical/SortingSpecial/udpComm_disp/_AddRemoveFromPool.st
